# B&R Automation Studio project Lab2_Conveyor
Automation Studio 4.5.2.102; Conveyor station; technology packages: Acp10Arnc0 5.2.1, mapp 5.2.1

## Configuration Distributor

CPU 5PP5CP.US15-02, AutomationRuntime D4.52, Build 4.1.2, Vc V4.52.0

### Task classes (Cpu.sw)
```
Cyclic#1 (cycle 2000 us, tolerance 0 us):
  ncsdcctrl <- ncsdcctrl.prg
  IOCtrl1 <- (binary)
  IOCtrl <- (binary)
Cyclic#4:
  Ejector <- Distributing.Machine.Ejector.prg
  SwivelDriv <- Distributing.Machine.SwivelDrive.prg
  AlarmCtrl <- Distributing.AlarmCtrl.prg
  MainCtrl <- Distributing.Machine.MainCtrl.prg
  Conveyor <- Distributing.Machine.Conveyor.Conveyor.prg
  VisCtrl <- Distributing.Visualization.VisCtrl.prg [disabled]
DataObjects: Acp10sys
NcDataObjects: gAxisDista <- Distributing.Machine.Conveyor.gAxisDistobj.gAxisDista.dob, gAxisDisti <- Distributing.Machine.Conveyor.gAxisDistobj.gAxisDisti.dob, acp10etxen <- acp10etxen.dob
VcDataObjects: VisuDi <- Distributing.Visualization.VisuDist.dob
Binaries: udbdef, TCData, arsvcreg, vccdt, vccbmp, vcfile, arial, vcrt, vcbclass, vccbtn, vcmgr, vcgclass, vcdsint, vcnet, vcptelo, vccline, vcpdihd, vcpfpp50, vcshared, vcclbox, vccscale, arialbd, vccnum, vcpdvnc, vcpdi855, vcpdsw, VisuDi01, vccshape, VisuDi02, vcctext, vcfntttf, vccovl, vcalarm, vcpdi815, VisuDi03, vcdsloc, vcpfmtcx, vctcal, arconfig, User, Config, ashwd, sysconf, ashwac, Role, asfw, iomap, OpcUaMap, Acp10map, acp10cfg
Libraries: AsOpcUac, runtime, AsOpcUas, asstring, brsystem, MpBase, MpCom, standard, sys_lib, Acp10par, NcGlobal, Acp10man, Acp10sdc, Acp10_MC, AsBrStr, MpAxis, asieccon, fileio, astime, dataobj, powerlnk, vcresman
```

### Hardware
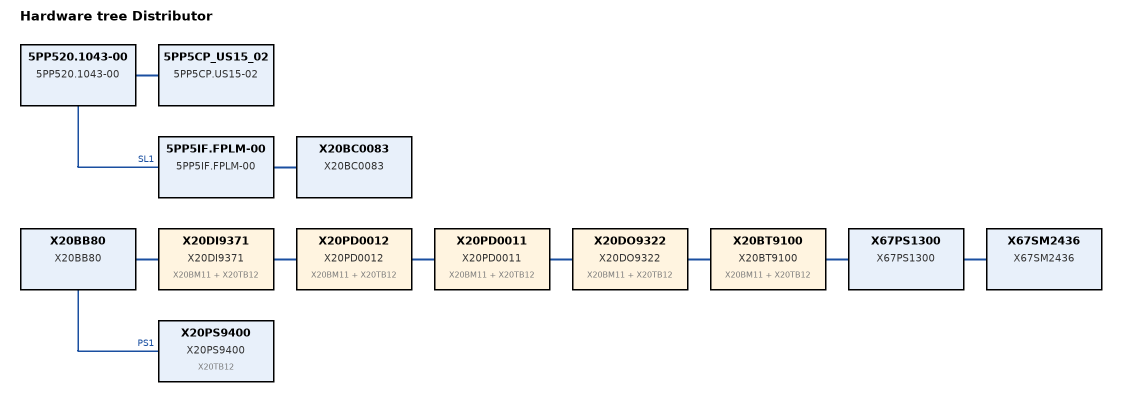
```
5PP520.1043-00 : 5PP520.1043-00 v2.0.3.1
  Connector IF3:
    ActivateDevice = 1
    Mode = Manual
    InternetAddress = 10.10.10.99
    SubnetMask = 255.255.255.0
    Vnc1
    VncVcObjectName1 = VisuDi
    VncKeyMappingFile1 = 
    VncRefreshRate1 = 250
  VcObjectName = VisuDi
5PP5CP_US15_02 : 5PP5CP.US15-02 v2.0.6.0  [SY -> 5PP520.1043-00.SY1]
  ConfigurationID = Lab2_Conveyor_Distributor
  TimerDeviceType = EPLX2X
  TimerDevice = 5PP5IF.FPLM-00.IF1
  TaskClassIdleTime = 2000
  Cyclic1Duration = 2000
  Cyclic1Tolerance = 0
  Cyclic1Output = 1
  ActivateOpcUa = 1
  OpcUaInformationModels_PV_Version = 1
5PP5IF.FPLM-00 : 5PP5IF.FPLM-00 v2.4.0.0  [SL -> 5PP520.1043-00.SL1]
X20BB80 : X20BB80 v1.0.2.0
X20BC0083 : X20BC0083 v2.7.0.0  [PLK1 -> 5PP5IF.FPLM-00.IF1 (NodeNumber=2) [Cable Type=PowerlinkCable, Length=10, Version=1.0.0.2]; SL -> X20BB80.SL1]
  Supervision = off
X20BM11 : X20BM11 v1.0.0.1  [X2X1 -> X20BB80.IF1]
X20BM11a : X20BM11 v1.0.0.1  [X2X1 -> X20BM11.X2X2]
X20BM11b : X20BM11 v1.0.0.1  [X2X1 -> X20BM11a.X2X2]
X20BM11c : X20BM11 v1.0.0.1  [X2X1 -> X20BM11b.X2X2]
X20BM11d : X20BM11 v1.0.0.1  [X2X1 -> X20BM11c.X2X2]
X20BT9100 : X20BT9100 v1.0.3.0  [SS1 -> X20TB12e.SS; SL -> X20BM11d.SL1]
  Supervision = off
X20DI9371 : X20DI9371 v1.0.2.0  [SS1 -> X20TB12a.SS; SL -> X20BM11.SL1]
  Supervision = off
X20DO9322 : X20DO9322 v1.0.3.0  [SS1 -> X20TB12d.SS; SL -> X20BM11c.SL1]
  Supervision = off
X20PD0011 : X20PD0011 v1.0.2.0  [SS1 -> X20TB12c.SS; SL -> X20BM11b.SL1]
  Supervision = off
X20PD0012 : X20PD0012 v1.0.2.0  [SS1 -> X20TB12b.SS; SL -> X20BM11a.SL1]
  Supervision = off
X20PS9400 : X20PS9400 v1.0.2.4  [SS1 -> X20TB12.SS; PS -> X20BB80.PS1]
  Supervision = off
X20TB12 : X20TB12 v1.0.0.0
X20TB12a : X20TB12 v1.0.0.0
X20TB12b : X20TB12 v1.0.0.0
X20TB12c : X20TB12 v1.0.0.0
X20TB12d : X20TB12 v1.0.0.0
X20TB12e : X20TB12 v1.0.0.0
X67PS1300 : X67PS1300 v1.0.0.0  [X2X1 -> X20BT9100.X2X1 [Cable Type=X2XCable, Length=10, Version=1.0.0.2]]
X67SM2436 : X67SM2436 v1.5.0.1  [X2X1 -> X67PS1300.X2X2 [Cable Type=X2XCable, Length=10, Version=1.0.0.2]]
  Supervision = off
  HoldingCurrent01 = 0
  RatedCurrent01 = 100
  MaximumCurrent01 = 160
  LatchSync01 = Stepper 1 latch value synchron (AB/R_1 latch value asynchron)
  LatchSync02 = Stepper 2 latch value synchron (AB/R_2 latch value asynchron)
  SCALE_ENCOD_INCR_r1 = 51200
  BothEndSwitchesAreNormallyOpen_r1 = on
```

### IoMap.iom - 5PP5CP_US15_02/IoMap.iom
```iecst
VAR_CONFIG
	Cyclic#1.gAxisDist_DrvIf.iLifeCnt AT %IB."X67SM2436".LifeCnt;
	Cyclic#1.gAxisDist_DrvIf.iDrvOK AT %IX."X67SM2436".DrvOk01;
	Cyclic#1.gAxisDist_DrvIf.oBoostCurrent AT %QX."X67SM2436".BoostCurrent01;
	Cyclic#1.gAxisDist_DrvIf.oStandStillCurrent AT %QX."X67SM2436".StandstillCurrent01;
	Cyclic#1.gAxisDist_DrvIf.oSetTime AT %QW."X67SM2436".SetTime01;
	Cyclic#1.gAxisDist_MotorStep0 AT %QW."X67SM2436".Motor1Step0;
	Cyclic#1.gAxisDist_DiDoIf.iLifeCntDriveEnable AT %IB."X67SM2436".LifeCnt;
	Cyclic#1.gAxisDist_DiDoIf.iLifeCntDriveReady AT %IB."X67SM2436".LifeCnt;
	Cyclic#1.gAxisDist_DiDoIf.iDriveReady AT %IX."X67SM2436".DrvOk01;
	Cyclic#1.gAxisDist_DiDoIf.oDriveEnable AT %QX."X67SM2436".DriveEnable01;
	Cyclic#1.gAxisDist_EncIf1.iLifeCnt AT %IB."X67SM2436".LifeCnt;
	Cyclic#1.gAxisDist_EncIf1.iEncOK AT %IX."X67SM2436".EncOk01;
	Cyclic#1.gAxisDist_EncIf1.iActPos AT %IW."X67SM2436".ActPos01;
	Cyclic#1.gAxisDist_EncIf1.iRefPulsePos AT %IW."X67SM2436".RefPulsePos01;
	Cyclic#1.gAxisDist_EncIf1.iRefPulseCnt AT %IB."X67SM2436".RefPulseCnt01;
	Cyclic#1.gAxisDist_EncIf1.iActTime AT %IW."X67SM2436".ActTime01;
	::gDistModuleOK.Interface AT %IX."5PP5IF.FPLM-00".ModuleOk;
	::gDistModuleOK.BusController AT %IX."X20BC0083".ModuleOk;
	::gDistModuleOK.PowerSupply AT %IX."X20PS9400".ModuleOk;
	::gDistModuleOK.DigitalInput AT %IX."X20DI9371".ModuleOk;
	::gDistModuleOK.PotentialDist0012 AT %IX."X20PD0012".ModuleOk;
	::gDistModuleOK.PotentialDist0011 AT %IX."X20PD0011".ModuleOk;
	::gDistModuleOK.DigitalOutput AT %IX."X20DO9322".ModuleOk;
	::gDistModuleOK.BusTransmitter AT %IX."X20BT9100".ModuleOk;
	::gDistModuleOK.StepperMotor AT %IX."X67SM2436".ModuleOk;
	::gDistHW.di.ProductGripped AT %IX."X20DI9371".DigitalInput04; (* *) (*Product gripped with suction*)
	::gDistHW.di.SwDrMagPos AT %IX."X20DI9371".DigitalInput05; (* *) (*Swivel drive in magazine position*)
	::gDistHW.di.SwDrConvPos AT %IX."X20DI9371".DigitalInput06; (* *) (*Swivel drive in conveyor position*)
	::gDistHW.di.MagEmpty AT %IX."X20DI9371".DigitalInput07; (* *) (*Magazine empty*)
	::gDistHW.di.SortStationFree AT %IX."X20DI9371".DigitalInput08; (* *) (*Sorting station free*)
	::gDistHW.do.EjCylPushProduct AT %QX."X20DO9322".DigitalOutput01; (* *) (*Ejecting cylinder push out product*)
	::gDistHW.do.Vacuum AT %QX."X20DO9322".DigitalOutput02; (* *) (*Vacuum on swivel drive*)
	::gDistHW.do.EjImpulse AT %QX."X20DO9322".DigitalOutput03; (* *) (*Ejection impulse on swivel drive*)
	::gDistHW.do.SwDrToMag AT %QX."X20DO9322".DigitalOutput04; (* *) (*Swivel drive to magazine*)
	::gDistHW.do.SwDrToConv AT %QX."X20DO9322".DigitalOutput05; (* *) (*Swivel drive to conveyor*)
	::gDistHW.di.EjCylRetracted AT %IX."X20DI9371".DigitalInput02; (* *) (*Ejecting cylinder retracted*)
	::gDistHW.di.EjCylExtended AT %IX."X20DI9371".DigitalInput03; (* *) (*Ejecting cylinder extended*)
	::gDistHW.di.PuckAtConvEnd AT %IX."X67SM2436".StatusInput01; (*Logical condition digital input 2, ABR2-A*) (*Conveyor - product on unloading position*) (*Logical condition digital input 4, ABR2-A*)
	::gDistHW.di.ConvStartVacant AT %IX."X67SM2436".StatusInput02; (*Logical condition digital input 1, ABR1-A*) (*Conveyor - product on starting position*)
END_VAR
```

### Acp10cfg.ncc - 5PP5CP_US15_02/Motion/Acp10cfg.ncc
```
NcConfiguration (Version=5.02.1, NcSwId=Acp10)
  ACP10CF1_typ:
    cnt_nettrc_rec_drive = 65535
    bufsize_trace_upload = 1200
    tc_nc_man_task = Cyclic #1
    glob_pv_as_ncobject = Yes
    ncsys_dl_broadcast = Yes
    ncsys_dl_acp_reset = Yes
    safemc_log_err_to_ax = Yes
    network_init:
      ncsw_init_execute = Yes
      automatic_execute = No
      node_nr_warning = Yes
      net_err_before_ncact = Yes
    nettrc:
      enter_parsecrec = Yes
      enter_ncaction = Yes
      save_ring_startidx = No
    cam_prof_download:
      cam_dat_dl_parallel = No
      tc_cam_dl_parallel = Task class for NC Manager task
    sdc_if[0]:
      if_name = SDC_IF1
      mc_broadcast_size = 800
      mc_broadcast_extdat = No
```

### Acp10map.ncm - 5PP5CP_US15_02/Motion/Acp10map.ncm
```
NcMapping (NcSwId=Acp10)
  NcObject gAxisDist (ModuleId=X67SM2436, ModuleAddress=SDC_IF1.ST1, Type=ncAXIS, Channel=1, AcoposSimulation=Off, InitParameter=gAxisDisti, AcoposParameter=gAxisDista, Disabled=FALSE, ModuleDisabled=FALSE)
  NcObject X67SM2436_ncAXIS2 (ModuleId=X67SM2436, ModuleAddress=SDC_IF1.ST2, Type=ncAXIS, Channel=1, AcoposSimulation=Off, Disabled=TRUE, ModuleDisabled=FALSE)
```

### Config.mpaxisbasic - 5PP5CP_US15_02/Motion/Config.mpaxisbasic
```
Element gAxisBasic (Type=mpaxisbasic)
  AxisConfiguration = AxisWithConfiguration
    Axis:
      BaseType = 2
      MeasurementUnit = 1
      PeriodSettings:
        Period = 108.0
      MovementLimits:
        VelocityPositive = 5000.0
        VelocityNegative = 5000.0
        Acceleration = 10000.0
        Deceleration = 10000.0
    Drive:
      Transformation:
        ReferenceDistance = 108.0
      Controller:
        LoopFilters:
          [0]
          [1]
          [2]
```

### Config_1.mpalarmxcore - 5PP5CP_US15_02/mappServices/Config_1.mpalarmxcore
```
Element gAlarmXCore_Dist (Type=mpalarmxcore)
  mapp.AlarmX.Core:
    Mapping:
      [0]:
        Alarm = Ejector Station - Cylinder Blocked
        [0] = Reaction
          Name = ErrorReaction
      [1]:
        Alarm = Swivel Arm - Motion Blocked
        [0] = Reaction
          Name = ErrorReaction
      [2]:
        Alarm = Conveyor - Puck Lost
        [0] = Reaction
          Name = ErrorReaction
      [3]:
        Alarm = Conveyor - Product Backlog
        [0] = Reaction
          Name = ErrorReaction
  mapp.AlarmX.Core.Configuration:
    [0]:
      Name = Ejector Station - Cylinder Blocked
      Message = Check for a backup in the ejector tray or a puck jammed in the magazine.
    [1]:
      Name = Swivel Arm - Motion Blocked
      Message = The Swivel Arm could not reach the requested position. Check for blockages.
    [2]:
      Name = Conveyor - Puck Lost
      Message = A puck is taking too long to reach the conveyor's end. Check for a lost puck or a sideways puck on the conveyor.
    [3]:
      Name = Conveyor - Product Backlog
      Message = There are too many unsorted pucks on the conveyor. Please remove excess pucks.
```

### Config_2.mpalarmxhistory - 5PP5CP_US15_02/mappServices/Config_2.mpalarmxhistory
```
Element gAlarmXHistory_Dist (Type=mpalarmxhistory)
```

## Configuration Sorter

CPU 5PP5CP.US15-02, AutomationRuntime D4.52, Build 4.1.2, Vc V4.52.0

### Task classes (Cpu.sw)
```
Cyclic#1 (cycle 2000 us, tolerance 0 us):
  ncsdcctrl <- ncsdcctrl.prg
Cyclic#4:
  MainCtrl <- Sorting.Machine.MainCtrl.prg
  OPCUAClien <- Sorting.OPCUA.OPCUAClient.prg [disabled]
  OPCUAConne <- Sorting.OPCUA.OPCUAConnect.prg [disabled]
  IOCtrl <- Sorting.Machine.IOCtrl.prg
  SortingSta <- Sorting.Machine.SortingStation.prg
  AlarmCtrl <- Sorting.AlarmCtrl.prg
  VisCtrl <- Sorting.Visualization.VisCtrl.prg
DataObjects: Acp10sys
NcDataObjects: gAxisSorta <- Sorting.gAxisSortobj.gAxisSorta.dob, gAxisSorti <- Sorting.gAxisSortobj.gAxisSorti.dob, acp10etxen <- acp10etxen.dob
VcDataObjects: VisuSo <- Sorting.Visualization.VisuSort.dob
Binaries: TCData, udbdef, vccdt, VisuSo02, vccbmp, vcfile, arial, vcrt, vcbclass, vccbtn, vcmgr, vcgclass, vcdsint, vcnet, vcptelo, vccline, vcpdihd, vcpfpp50, vcshared, vcclbox, vccscale, arialbd, vccnum, vcpdvnc, vcpdi855, vcpdsw, vccshape, vcctext, vcfntttf, vccovl, vcalarm, vcpdi815, arsvcreg, vcdsloc, vcpfmtcx, vctcal, VisuSo01, VisuSo03, vcchspot, Config_2, Config_1, OpcUaMap, ashwd, Role, User, sysconf, ashwac, asfw, arconfig, Config, iomap, Acp10map, acp10cfg, vcpkat, vcpfar00
Libraries: Acp10sdc, Acp10man, Acp10_MC, sys_lib, brsystem, AsBrStr, operator, runtime, astime, AsIecCon, AsOpcUac, AsOpcUas, asstring, MpCom, MpBase, standard, Acp10par, NcGlobal, MpAxis, MpAlarmX, fileio, powerlnk, vcresman, dataobj, areventlog
```

### Hardware
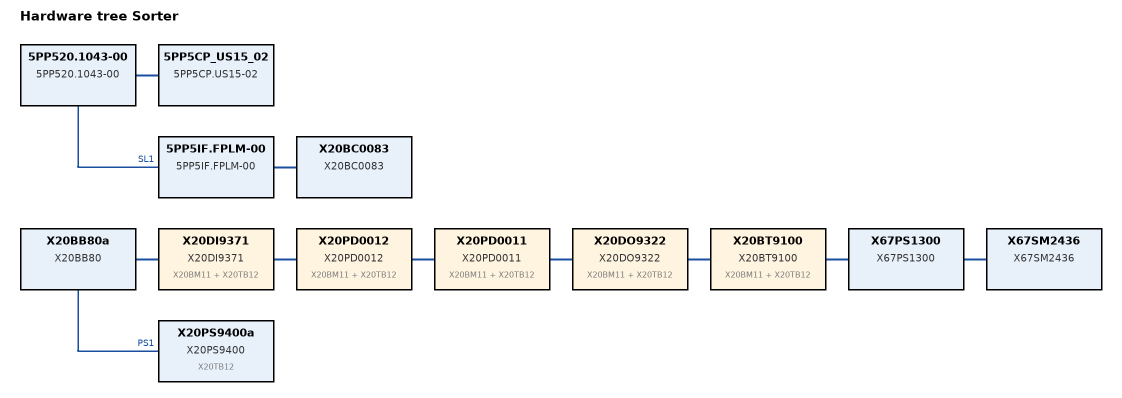
```
5PP520.1043-00 : 5PP520.1043-00 v2.0.3.1
  Connector IF3:
    ActivateDevice = 1
    Mode = Manual
    InternetAddress = 10.10.10.100
    SubnetMask = 255.255.255.0
    Vnc1
    VncVcObjectName1 = VisuSo
    VncKeyMappingFile1 = 
    VncRefreshRate1 = 250
  VcObjectName = VisuSo
5PP5CP_US15_02 : 5PP5CP.US15-02 v2.0.6.0  [SY -> 5PP520.1043-00.SY1]
  ConfigurationID = Lab2_Conveyor_Sorter
  TimerDeviceType = EPLX2X
  TimerDevice = 5PP5IF.FPLM-00.IF1
  TaskClassIdleTime = 2000
  Cyclic1Duration = 2000
  Cyclic1Tolerance = 0
  Cyclic1Output = 1
  ActivateOpcUa = 1
  OpcUaInformationModels_PV_Version = 1
5PP5IF.FPLM-00 : 5PP5IF.FPLM-00 v2.4.0.0  [SL -> 5PP520.1043-00.SL1]
X20BB80a : X20BB80 v1.0.2.0
X20BC0083 : X20BC0083 v2.7.0.0  [PLK1 -> 5PP5IF.FPLM-00.IF1 [Cable Type=PowerlinkCable, Length=10, Version=1.0.0.2]; SL -> X20BB80a.SL1]
X20BM11 : X20BM11 v1.0.0.1  [X2X1 -> X20BB80a.IF1]
X20BM11a : X20BM11 v1.0.0.1  [X2X1 -> X20BM11.X2X2]
X20BM11b : X20BM11 v1.0.0.1  [X2X1 -> X20BM11a.X2X2]
X20BM11c : X20BM11 v1.0.0.1  [X2X1 -> X20BM11b.X2X2]
X20BM11d : X20BM11 v1.0.0.1  [X2X1 -> X20BM11c.X2X2]
X20BT9100 : X20BT9100 v1.0.3.0  [SS1 -> X20TB12e.SS; SL -> X20BM11d.SL1]
X20DI9371 : X20DI9371 v1.0.2.0  [SS1 -> X20TB12b.SS; SL -> X20BM11.SL1]
X20DO9322 : X20DO9322 v1.0.3.0  [SS1 -> X20TB12d.SS; SL -> X20BM11c.SL1]
X20PD0011 : X20PD0011 v1.0.2.0  [SS1 -> X20TB12c.SS; SL -> X20BM11b.SL1]
X20PD0012 : X20PD0012 v1.0.2.0  [SS1 -> X20TB12.SS; SL -> X20BM11a.SL1]
X20PS9400a : X20PS9400 v1.0.2.4  [SS1 -> X20TB12a.SS; PS -> X20BB80a.PS1]
X20TB12 : X20TB12 v1.0.0.0
X20TB12a : X20TB12 v1.0.0.0
X20TB12b : X20TB12 v1.0.0.0
X20TB12c : X20TB12 v1.0.0.0
X20TB12d : X20TB12 v1.0.0.0
X20TB12e : X20TB12 v1.0.0.0
X67PS1300 : X67PS1300 v1.0.0.0  [X2X1 -> X20BT9100.X2X1 [Cable Type=X2XCable, Length=10, Version=1.0.0.2]]
X67SM2436 : X67SM2436 v1.5.0.1  [X2X1 -> X67PS1300.X2X2 [Cable Type=X2XCable, Length=10, Version=1.0.0.2]]
  Supervision = off
  HoldingCurrent01 = 0
  RatedCurrent01 = 80
  MaximumCurrent01 = 160
  LatchSync01 = Stepper 1 latch value synchron (AB/R_1 latch value asynchron)
  SCALE_ENCOD_INCR_r1 = 51200
```

### IoMap.iom - 5PP5CP_US15_02/IoMap.iom
```iecst
VAR_CONFIG
	Cyclic#1.gAxisSort_DrvIf.iLifeCnt AT %IB."X67SM2436".LifeCnt;
	Cyclic#1.gAxisSort_DrvIf.iDrvOK AT %IX."X67SM2436".DrvOk01;
	Cyclic#1.gAxisSort_DrvIf.oBoostCurrent AT %QX."X67SM2436".BoostCurrent01;
	Cyclic#1.gAxisSort_DrvIf.oStandStillCurrent AT %QX."X67SM2436".StandstillCurrent01;
	Cyclic#1.gAxisSort_DrvIf.oSetTime AT %QW."X67SM2436".SetTime01;
	Cyclic#1.gAxisSort_MotorStep0 AT %QW."X67SM2436".Motor1Step0;
	Cyclic#1.gAxisSort_DiDoIf.iLifeCntDriveEnable AT %IB."X67SM2436".LifeCnt;
	Cyclic#1.gAxisSort_DiDoIf.iLifeCntDriveReady AT %IB."X67SM2436".LifeCnt;
	Cyclic#1.gAxisSort_DiDoIf.iDriveReady AT %IX."X67SM2436".DrvOk01;
	Cyclic#1.gAxisSort_DiDoIf.oDriveEnable AT %QX."X67SM2436".DriveEnable01;
	Cyclic#1.gAxisSort_EncIf1.iLifeCnt AT %IB."X67SM2436".LifeCnt;
	Cyclic#1.gAxisSort_EncIf1.iEncOK AT %IX."X67SM2436".EncOk01;
	Cyclic#1.gAxisSort_EncIf1.iActPos AT %IW."X67SM2436".ActPos01;
	Cyclic#1.gAxisSort_EncIf1.iRefPulsePos AT %IW."X67SM2436".RefPulsePos01;
	Cyclic#1.gAxisSort_EncIf1.iRefPulseCnt AT %IB."X67SM2436".RefPulseCnt01;
	Cyclic#1.gAxisSort_EncIf1.iActTime AT %IW."X67SM2436".ActTime01;
	::gSortHW.do.ExtendSwitch1 AT %QX."X20DO9322".DigitalOutput02; (* *) (*Extend switch 1*)
	::gSortHW.do.ExtendSwitch2 AT %QX."X20DO9322".DigitalOutput03; (* *) (*Extend switch 2*)
	::gSortHW.do.RetractStopper AT %QX."X20DO9322".DigitalOutput04; (* *) (*Retract stopper*)
	::gSortHW.di.ProductAvailable AT %IX."X20DI9371".DigitalInput01; (* *) (*Product available*)
	::gSortHW.di.Metallic AT %IX."X20DI9371".DigitalInput02; (* *) (*Metallic product*)
	::gSortHW.di.NotBlack AT %IX."X20DI9371".DigitalInput03; (* *) (*Product is not black*)
	::gSortHW.di.LaneFull AT %IX."X20DI9371".DigitalInput04; (* *) (*Lane full*)
	::gSortHW.di.Switch1Retracted AT %IX."X20DI9371".DigitalInput05; (* *) (*Switch 1 retracted*)
	::gSortHW.di.Switch1Extended AT %IX."X20DI9371".DigitalInput06; (* *) (*Switch 1 extended*)
	::gSortHW.di.Switch2Retracted AT %IX."X20DI9371".DigitalInput07; (* *) (*Switch 2 retracted*)
	::gSortHW.di.Switch2Extended AT %IX."X20DI9371".DigitalInput08; (* *) (*Switch 2 extended*)
	::gSortModuleOK.Interface AT %IX."5PP5IF.FPLM-00".ModuleOk;
	::gSortModuleOK.BusController AT %IX."X20BC0083".ModuleOk;
	::gSortModuleOK.PowerSupply AT %IX."X20PS9400a".ModuleOk;
	::gSortModuleOK.DigitalInput AT %IX."X20DI9371".ModuleOk;
	::gSortModuleOK.PotentialDist0012 AT %IX."X20PD0012".ModuleOk;
	::gSortModuleOK.PotentialDist0011 AT %IX."X20PD0011".ModuleOk;
	::gSortModuleOK.DigitalOutput AT %IX."X20DO9322".ModuleOk;
	::gSortModuleOK.BusTransmitter AT %IX."X20BT9100".ModuleOk;
	::gSortModuleOK.StepperMotor AT %IX."X67SM2436".ModuleOk;
END_VAR
```

### Acp10cfg.ncc - 5PP5CP_US15_02/Motion/Acp10cfg.ncc
```
NcConfiguration (Version=5.02.1, NcSwId=Acp10)
  ACP10CF1_typ:
    cnt_nettrc_rec_drive = 65535
    bufsize_trace_upload = 1200
    tc_nc_man_task = Cyclic #1
    glob_pv_as_ncobject = Yes
    ncsys_dl_broadcast = Yes
    ncsys_dl_acp_reset = Yes
    safemc_log_err_to_ax = Yes
    network_init:
      ncsw_init_execute = Yes
      automatic_execute = No
      node_nr_warning = Yes
      net_err_before_ncact = Yes
    nettrc:
      enter_parsecrec = Yes
      enter_ncaction = Yes
      save_ring_startidx = Yes
    cam_prof_download:
      cam_dat_dl_parallel = No
      tc_cam_dl_parallel = Task class for NC Manager task
    sdc_if[0]:
      if_name = SDC_IF1
      mc_broadcast_size = 800
      mc_broadcast_extdat = No
```

### Acp10map.ncm - 5PP5CP_US15_02/Motion/Acp10map.ncm
```
NcMapping (NcSwId=Acp10, DisabledNodesAreHidden=False)
  NcObject gAxisSort (ModuleId=X67SM2436, ModuleAddress=SDC_IF1.ST1, Type=ncAXIS, Channel=1, AcoposSimulation=Off, InitParameter=gAxisSorti, AcoposParameter=gAxisSorta, Disabled=FALSE, ModuleDisabled=FALSE)
  NcObject X67SM2436_ncAXIS2 (ModuleId=X67SM2436, ModuleAddress=SDC_IF1.ST2, Type=ncAXIS, Channel=1, AcoposSimulation=Off, Disabled=TRUE, ModuleDisabled=FALSE)
```

### Config.mpaxisbasic - 5PP5CP_US15_02/Motion/Config.mpaxisbasic
```
Element gAxisBasic (Type=mpaxisbasic)
  AxisConfiguration = AxisWithConfiguration
    Axis:
      BaseType = 2
      MeasurementUnit = 1
      MeasurementResolution = 1
      PeriodSettings:
        Period = 150
      MovementLimits:
        VelocityPositive = 10000
        VelocityNegative = 10000
        Acceleration = 50000
        Deceleration = 50000
    Drive:
      Transformation:
        ReferenceDistance = 150
      Controller:
        LoopFilters:
          [0]
          [1]
          [2]
```

### Config_1.mpalarmxcore - 5PP5CP_US15_02/mappServices/Config_1.mpalarmxcore
```
Element gAlarmXCore_Sort (Type=mpalarmxcore)
  mapp.AlarmX.Core.Configuration:
    [0]:
      Name = Lane1Full
      Message = Lane 1 is full.
      Code = 1
    [1]:
      Name = Lane2Full
      Message = Lane 2 is full.
      Code = 2
    [2]:
      Name = Lane3Full
      Message = Lane 3 is full.
      Code = 3
    [3]:
      Name = NoProductAvail
      Message = There is no product available.
      Code = 4
    [4]:
      Name = SwitchStuck
      Message = The switch is stuck.
      Code = 5
    [5]:
      Name = PuckMissing
      Message = No product detected.
      Code = 6
    [6]:
      Name = Axis
      Message = Axis error.
      Code = 7
    [7]:
      Name = CheckHW
      Message = Hardware module not OK.
      Code = 8
    [8]:
      Name = CheckMachine
      Message = Machine error.
      Code = 9
```

### Config_2.mpalarmxhistory - 5PP5CP_US15_02/mappServices/Config_2.mpalarmxhistory
```
Element gAlarmXHistory_Sort (Type=mpalarmxhistory)
```

## Logical view

Binary libraries used (declarations not repeated): operator, runtime, astime, AsIecCon, AsOpcUac, AsOpcUas, asstring, brsystem, MpCom 5.02.1, standard, sys_lib, AsBrStr, MpAxis 1.65.0, MpBase 5.02.0, NcGlobal, Acp10_MC, Acp10man, Acp10par, Acp10sdc, MpAlarmX 5.02.1

### Global.var - Global variables
```iecst
VAR
	gAxisDist : ACP10AXIS_typ; (*Axis variable distributor*)
	gAxisDist_HW : SdcHwCfg_typ := (0); (*Axis variable distributor*)
	gAxisDist_DrvIf : SdcDrvIf16_typ := (0); (*Axis variable distributor*)
	gAxisDist_EncIf1 : SdcEncIf16_typ := (0); (*Axis variable distributor*)
	gAxisDist_DiDoIf : SdcDiDoIf_typ := (0); (*Axis variable distributor*)
	gAxisDist_MotorStep0 : INT := 0; (*Axis variable distributor*)
	gAxisSort : ACP10AXIS_typ; (*Axis variable sorter*)
	gAxisSort_HW : SdcHwCfg_typ := (0); (*Axis variable sorter*)
	gAxisSort_DrvIf : SdcDrvIf16_typ := (0); (*Axis variable sorter*)
	gAxisSort_EncIf1 : SdcEncIf16_typ := (0); (*Axis variable sorter*)
	gAxisSort_DiDoIf : SdcDiDoIf_typ := (0); (*Axis variable sorter*)
	gAxisSort_MotorStep0 : INT := 0; (*Axis variable sorter*)
END_VAR
```

### Program Logical/ncsdcctrl (IEC) - ncsdcctrl

#### ncsdcctrl.var
```iecst
VAR
	gAxisDist_oSetPosOld : INT := 0;
	gAxisSort_oSetPosOld : INT := 0;
END_VAR
```

#### ncsdcctrlCyclic.st
```iecst
PROGRAM _CYCLIC

(* ### BEGIN gAxisDist ### *)

(* life counter emulation of digital inputs *)
       gAxisDist_DiDoIf.iLifeCntReference := gAxisDist_DiDoIf.iLifeCntReference + 1;
       gAxisDist_DiDoIf.iLifeCntNegHwEnd  := gAxisDist_DiDoIf.iLifeCntNegHwEnd  + 1;
       gAxisDist_DiDoIf.iLifeCntPosHwEnd  := gAxisDist_DiDoIf.iLifeCntPosHwEnd  + 1;

(* default function model of ACOPOSmicro: convert absolute steps to delta steps - overflow save delta calculation *)
       gAxisDist_MotorStep0 := gAxisDist_DrvIf.oSetPos - gAxisDist_oSetPosOld;
       gAxisDist_oSetPosOld := gAxisDist_DrvIf.oSetPos;

(* ### END gAxisDist ### *)

(* ### BEGIN gAxisSort ### *)

(* life counter emulation of digital inputs *)
       gAxisSort_DiDoIf.iLifeCntReference := gAxisSort_DiDoIf.iLifeCntReference + 1;
       gAxisSort_DiDoIf.iLifeCntNegHwEnd  := gAxisSort_DiDoIf.iLifeCntNegHwEnd  + 1;
       gAxisSort_DiDoIf.iLifeCntPosHwEnd  := gAxisSort_DiDoIf.iLifeCntPosHwEnd  + 1;

(* default function model of ACOPOSmicro: convert absolute steps to delta steps - overflow save delta calculation *)
       gAxisSort_MotorStep0 := gAxisSort_DrvIf.oSetPos - gAxisSort_oSetPosOld;
       gAxisSort_oSetPosOld := gAxisSort_DrvIf.oSetPos;

(* ### END gAxisSort ### *)

END_PROGRAM
```

#### ncsdcctrlInit.st
```iecst
PROGRAM _INIT

(* ### BEGIN gAxisDist ### *)

(* initialize general interfaces *)
       gAxisDist.size := gAxisDist.size;
       gAxisDist_HW.DrvIf_Typ := ncSDC_DRVSM16;
       brsstrcpy( ADR(gAxisDist_HW.DrvIf_Name[0]), ADR('gAxisDist_DrvIf') );
       gAxisDist_HW.DiDoIf_Typ := ncSDC_DIDO;
       brsstrcpy( ADR(gAxisDist_HW.DiDoIf_Name[0]), ADR('gAxisDist_DiDoIf') );
       gAxisDist_HW.EncIf1_Typ := ncSDC_ENC16;
       brsstrcpy( ADR(gAxisDist_HW.EncIf1_Name[0]), ADR('gAxisDist_EncIf1') );
       gAxisDist_EncIf1.iLifeCnt := gAxisDist_EncIf1.iLifeCnt;

(* initialize old-value for delta step calculation *)
       gAxisDist_oSetPosOld := gAxisDist_DrvIf.oSetPos;

(* ### END gAxisDist ### *)

(* ### BEGIN gAxisSort ### *)

(* initialize general interfaces *)
       gAxisSort.size := gAxisSort.size;
       gAxisSort_HW.DrvIf_Typ := ncSDC_DRVSM16;
       brsstrcpy( ADR(gAxisSort_HW.DrvIf_Name[0]), ADR('gAxisSort_DrvIf') );
       gAxisSort_HW.DiDoIf_Typ := ncSDC_DIDO;
       brsstrcpy( ADR(gAxisSort_HW.DiDoIf_Name[0]), ADR('gAxisSort_DiDoIf') );
       gAxisSort_HW.EncIf1_Typ := ncSDC_ENC16;
       brsstrcpy( ADR(gAxisSort_HW.EncIf1_Name[0]), ADR('gAxisSort_EncIf1') );
       gAxisSort_EncIf1.iLifeCnt := gAxisSort_EncIf1.iLifeCnt;

(* initialize old-value for delta step calculation *)
       gAxisSort_oSetPosOld := gAxisSort_DrvIf.oSetPos;

(* ### END gAxisSort ### *)

END_PROGRAM
```


### Package Logical/Distributing - Distributor configuration

### DistGlobal.typ - Package global types
```iecst
TYPE
	gDistHW_type : 	STRUCT  (*Hardware IO types for distributor*)
		di : diDist_type; (*Digital inputs for distributor*)
		do : doDist_type; (*Digital outputs for distributor*)
	END_STRUCT;
	diDist_type : 	STRUCT  (*Digital inputs for distributor*)
		EjCylExtended : BOOL; (*Ejecting cylinder extended*)
		EjCylRetracted : BOOL; (*Ejecting cylinder retracted*)
		ProductGripped : BOOL; (*Product gripped with suction*)
		SwDrMagPos : BOOL; (*Swivel drive in magazine position*)
		SwDrConvPos : BOOL; (*Swivel drive in conveyor position*)
		MagEmpty : BOOL; (*Magazine empty*)
		SortStationFree : BOOL; (*Sorting station free*)
		ConvStartVacant : BOOL; (*Conveyor - product on starting position*)
		PuckAtConvEnd : BOOL; (*Conveyor - product on unloading position*)
	END_STRUCT;
	doDist_type : 	STRUCT  (*Digital outputs for distributor*)
		EjCylPushProduct : BOOL; (*Ejecting cylinder push out product*)
		Vacuum : BOOL; (*Vacuum on swivel drive*)
		EjImpulse : BOOL; (*Ejection impulse on swivel drive*)
		SwDrToMag : BOOL; (*Swivel drive to magazine*)
		SwDrToConv : BOOL; (*Swivel drive to conveyor*)
	END_STRUCT;
	gDistModuleOK_type : 	STRUCT  (*Distributor module statuses*)
		Interface : BOOL; (*5PP5IF.FPLM-00 status*)
		BusController : BOOL; (*X20BC0083 status*)
		PowerSupply : BOOL; (*X20PS9400 status*)
		DigitalInput : BOOL; (*X20DI9371 status*)
		PotentialDist0012 : BOOL; (*X20PD0012 status*)
		PotentialDist0011 : BOOL; (*X20PD0011 status*)
		DigitalOutput : BOOL; (*X20DO9322 status*)
		BusTransmitter : BOOL; (*X20BT9100 status*)
		StepperMotor : BOOL; (*X67SM2436 status*)
	END_STRUCT;
END_TYPE
```

### DistGlobal.var - Package global variables
```iecst
VAR
	gDistHW : gDistHW_type; (*Control variable for hardware IO types for distributor*)
	gDistModuleOK : gDistModuleOK_type; (*Control variable for distributor module statuses*)
END_VAR
```

- Visualisation Logical/Distributing/Visualization (not shown)

### Package Logical/Distributing/Machine - Distributing machine functionality

### Package Logical/Distributing/Machine/Conveyor - Contains conveyor task and relevant motion items

### Package Logical/Distributing/Machine/Conveyor/gAxisDistobj - gAxisDistobj

### Data object Logical/Distributing/Machine/Conveyor/gAxisDistobj/gAxisDista (Apt)

#### gAxisDista.apt
```
AcoposParameterTable:
  Root Parameters:
    64232 = 51200 (Name=SM_SCALE_STEP)
    64233 = 1000 (Name=SM_SCALE_LOAD_UNITS)
    64234 = 1 (Name=SM_SCALE_LOAD_MOTREV)
    230 = PCTRL_S_SET (Name=PCTRL_S_ACT_PARID)  // CTRL Position controller: Actual encoder position parameter ID
```

### Data object Logical/Distributing/Machine/Conveyor/gAxisDistobj/gAxisDisti (Ax)

#### gAxisDisti.ax
```
InitParameter (Version=5.02.1, NcSwId=Acp10)
  ACP10AXIS_typ:
    dig_in:
      level:
        reference = ncACTIV_HI
        pos_hw_end = ncACTIV_HI
        neg_hw_end = ncACTIV_HI
        trigger1 = ncACTIV_HI
        trigger2 = ncACTIV_HI
    encoder_if:
      parameter:
        count_dir = ncSTANDARD
        scaling:
          load:
            units = 1000
            rev_motor = 1
    limit:
      parameter:
        v_pos = 3000.0
        v_neg = 3000.0
        a1_pos = 6000.0
        a2_pos = 6000.0
        a1_neg = 6000.0
        a2_neg = 6000.0
        t_jolt = 0
        t_in_pos = 0
        pos_sw_end = 2000000000
        neg_sw_end = -2000000000
        ds_warning = 500
        ds_stop = 1000
        a_stop = 1.0e30
        dv_stop = 0
        dv_stop_mode = ncOFF
    controller:
      mode = ncPOSITION
      position:
        kv = 50
        tn = 0
        t_predict = 0.01
        t_total = 0.01
        p_max = 1.0e30
        i_max = 0
      speed:
        kv = 2.0
        tn = 0
        t_filter = 0.0
        isq_filter1:
          type = ncOFF
          a0 = 0.0
          a1 = 0.0
          b0 = 0.0
          b1 = 0.0
          b2 = 0.0
          c0_par_id = 0
          c1_par_id = 0
        isq_filter2:
          type = ncOFF
          a0 = 0.0
          a1 = 0.0
          b0 = 0.0
          b1 = 0.0
          b2 = 0.0
          c0_par_id = 0
          c1_par_id = 0
        isq_filter3:
          type = ncOFF
          a0 = 0.0
          a1 = 0.0
          b0 = 0.0
          b1 = 0.0
          b2 = 0.0
          c0_par_id = 0
          c1_par_id = 0
      uf:
        type = ncLINEAR + ncCORRECTION
        auto_config = ncMOTOR_PAR
        u0 = 0
        un = 0
        fn = 50.0
        k_f_slip = 0
      ff:
        torque_load = 0.0
        torque_pos = 0.0
        torque_neg = 0.0
        kv_torque = 0.0
        inertia = 0.0
        t_filter_a = 0.0
    move:
      stop:
        parameter[0]:
          decel_ramp = ncA_LIMIT
          controller = ncON
        parameter[1]:
          decel_ramp = ncA_LIMIT
          controller = ncON
        parameter[2]:
          decel_ramp = ncA_LIMIT
          controller = ncON
        parameter[3]:
          decel_ramp = ncA_LIMIT
          controller = ncON
        quickstop:
          decel_ramp = ncA_LIMIT
          t_jolt = 0
        drive_error:
          decel_ramp = ncA_LIMIT
      homing:
        parameter:
          s = 0
          v_switch = 5000
          v_trigger = 500
          a = 50000
          mode = ncDIRECT
          edge_sw = ncPOSITIVE
          start_dir = ncPOSITIVE
          trigg_dir = ncPOSITIVE
          ref_pulse = ncOFF
          fix_dir = ncOFF
          tr_s_block = 0
          torque_lim = 0
          ds_block = 0
          ds_stop = 0
      basis:
        parameter:
          v_pos = 5000
          v_neg = 5000
          a1_pos = 50000
          a2_pos = 50000
          a1_neg = 50000
          a2_neg = 50000
    message:
      text:
        parameter:
          format = ncBREAK
          columns = 80
          data_modul = acp10etxen
```

### Program Logical/Distributing/Machine/Conveyor/Conveyor (IEC)

#### Cyclic.ld - Cyclic code
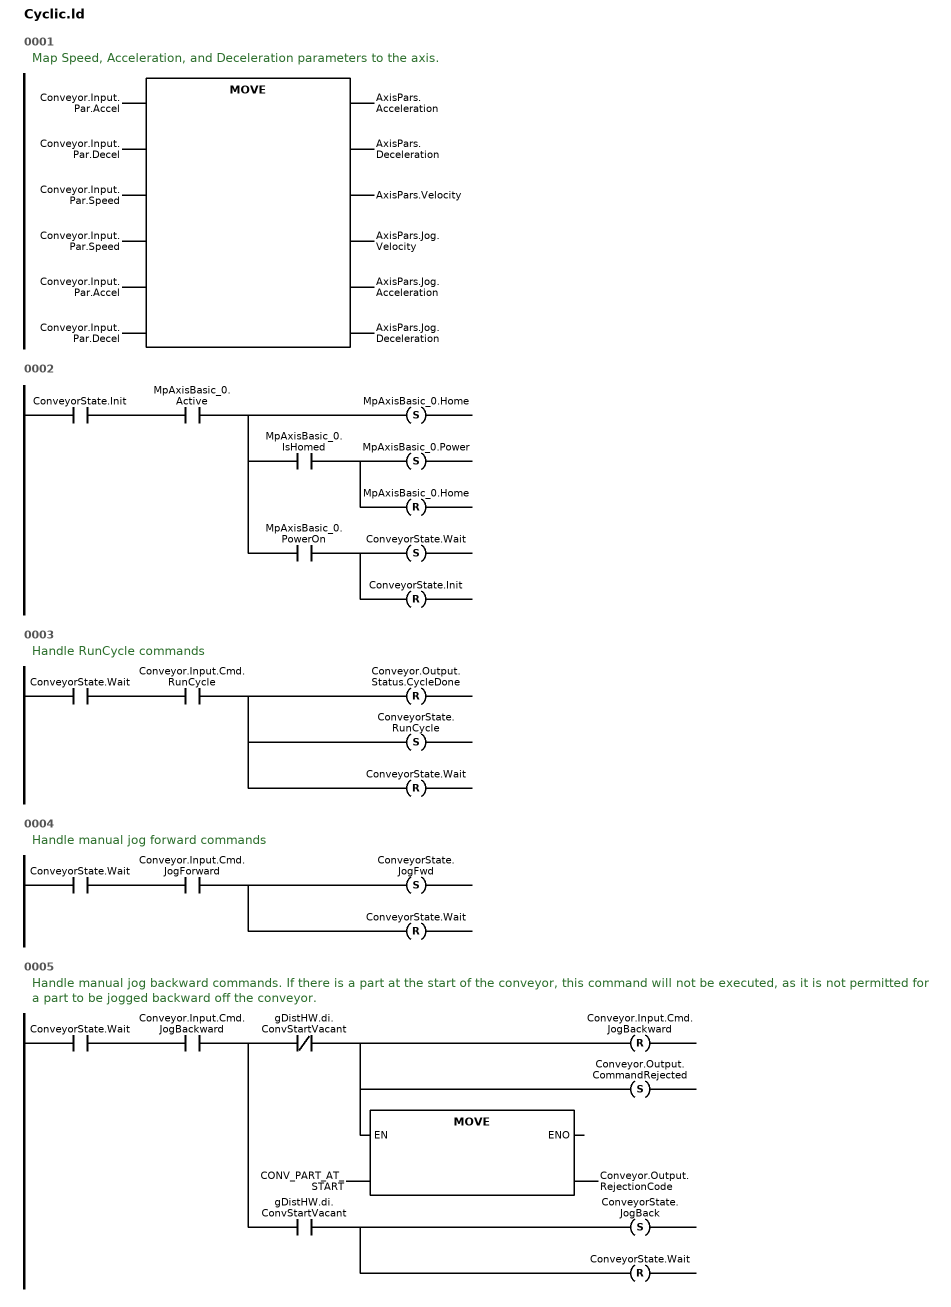
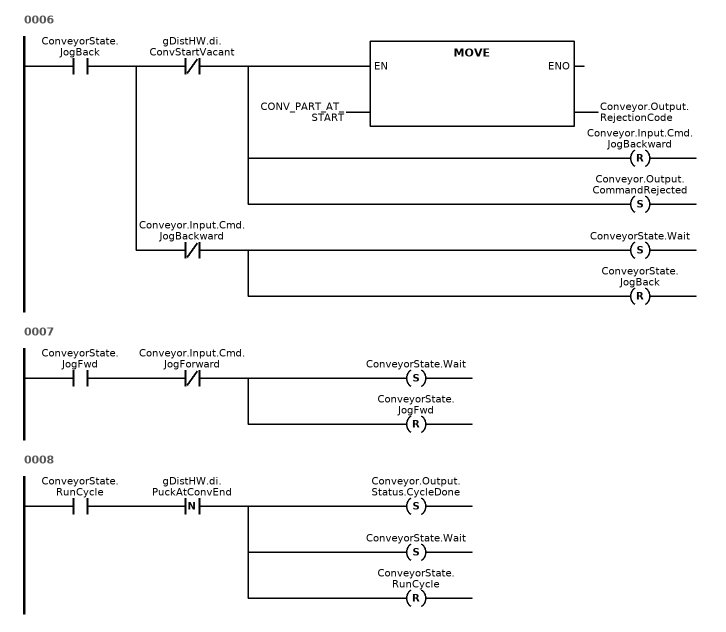
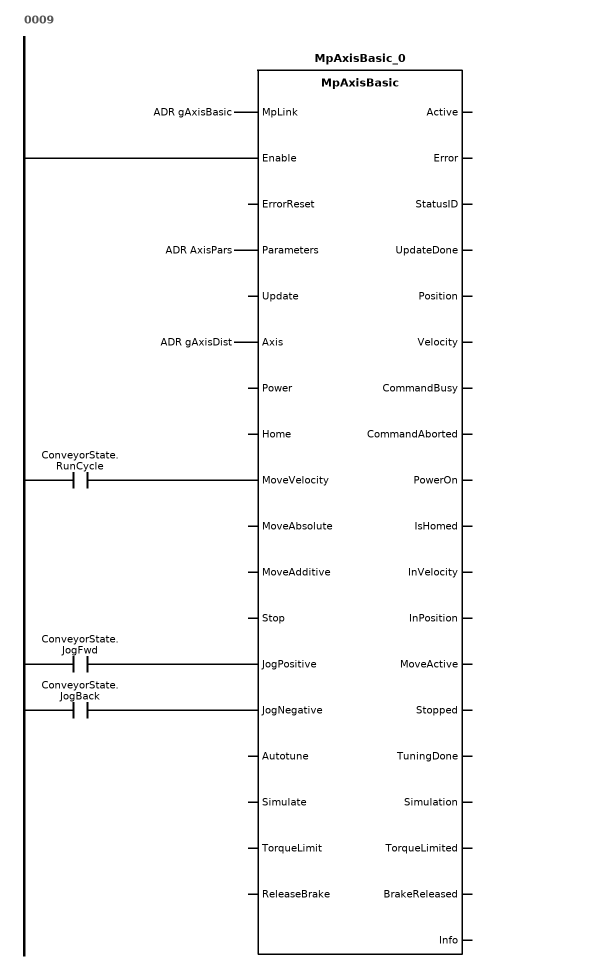
Ladder, written as Structured Text:
```iecst
(*********************************************************************************
 * Copyright:
 * Author:
 * Created:   	March 8, 2019/12:39 PM
 * Description:
 *********************************************************************************)
PROGRAM _CYCLIC
VAR
    _p1 : BOOL;
    _p2 : BOOL;
    _p3 : BOOL;
    _p4 : BOOL;
    _p5 : BOOL;
    _p6 : BOOL;
    _p7 : BOOL;
    _p8 : BOOL;
    _e9 : F_TRIG;
    _p10 : BOOL;
END_VAR
(* Network 1: Map Speed, Acceleration, and Deceleration parameters to the axis. *)
AxisPars.Acceleration := Conveyor.Input.Par.Accel;
AxisPars.Deceleration := Conveyor.Input.Par.Decel;
AxisPars.Velocity := Conveyor.Input.Par.Speed;
AxisPars.Jog.Velocity := Conveyor.Input.Par.Speed;
AxisPars.Jog.Acceleration := Conveyor.Input.Par.Accel;
AxisPars.Jog.Deceleration := Conveyor.Input.Par.Decel;

(* Network 2 *)
_p1 := ConveyorState.Init AND MpAxisBasic_0.Active;
IF ConveyorState.Init AND MpAxisBasic_0.Active THEN MpAxisBasic_0.Home := TRUE; END_IF;
_p2 := _p1 AND MpAxisBasic_0.IsHomed;
IF _p1 AND MpAxisBasic_0.IsHomed THEN MpAxisBasic_0.Power := TRUE; END_IF;
IF _p2 THEN MpAxisBasic_0.Home := FALSE; END_IF;
IF _p1 AND MpAxisBasic_0.PowerOn THEN
    ConveyorState.Wait := TRUE;
    ConveyorState.Init := FALSE;
END_IF;

(* Network 3: Handle RunCycle commands *)
_p3 := ConveyorState.Wait AND Conveyor.Input.Cmd.RunCycle;
IF _p3 THEN
    Conveyor.Output.Status.CycleDone := FALSE;
    ConveyorState.RunCycle := TRUE;
    ConveyorState.Wait := FALSE;
END_IF;

(* Network 4: Handle manual jog forward commands *)
_p4 := ConveyorState.Wait AND Conveyor.Input.Cmd.JogForward;
IF _p4 THEN
    ConveyorState.JogFwd := TRUE;
    ConveyorState.Wait := FALSE;
END_IF;

(* Network 5: Handle manual jog backward commands. If there is a part at the start of the conveyor, this command will not be executed, as it is not permitted for a part to be jogged backward off the conveyor. *)
_p5 := ConveyorState.Wait AND Conveyor.Input.Cmd.JogBackward;
IF _p5 AND NOT gDistHW.di.ConvStartVacant THEN
    Conveyor.Input.Cmd.JogBackward := FALSE;
    Conveyor.Output.CommandRejected := TRUE;
    Conveyor.Output.RejectionCode := CONV_PART_AT_START;
END_IF;
IF _p5 AND gDistHW.di.ConvStartVacant THEN
    ConveyorState.JogBack := TRUE;
    ConveyorState.Wait := FALSE;
END_IF;

(* Network 6 *)
_p6 := ConveyorState.JogBack AND NOT gDistHW.di.ConvStartVacant;
IF _p6 THEN
    Conveyor.Output.RejectionCode := CONV_PART_AT_START;
    Conveyor.Input.Cmd.JogBackward := FALSE;
    Conveyor.Output.CommandRejected := TRUE;
END_IF;
_p7 := ConveyorState.JogBack AND NOT Conveyor.Input.Cmd.JogBackward;
IF _p7 THEN
    ConveyorState.Wait := TRUE;
    ConveyorState.JogBack := FALSE;
END_IF;

(* Network 7 *)
_p8 := ConveyorState.JogFwd AND NOT Conveyor.Input.Cmd.JogForward;
IF _p8 THEN
    ConveyorState.Wait := TRUE;
    ConveyorState.JogFwd := FALSE;
END_IF;

(* Network 8 *)
_e9(CLK := gDistHW.di.PuckAtConvEnd);
IF ConveyorState.RunCycle AND _e9.Q THEN Conveyor.Output.Status.CycleDone := TRUE; END_IF;
_p10 := ConveyorState.RunCycle AND _e9.Q;
IF ConveyorState.RunCycle AND _e9.Q THEN ConveyorState.Wait := TRUE; END_IF;
IF _p10 THEN ConveyorState.RunCycle := FALSE; END_IF;

(* Network 9 *)
MpAxisBasic_0(MpLink := ADR(gAxisBasic), Enable := TRUE, Parameters := ADR(AxisPars), Axis := ADR(gAxisDist), MoveVelocity := ConveyorState.RunCycle, JogPositive := ConveyorState.JogFwd, JogNegative := ConveyorState.JogBack);
END_PROGRAM
```

#### Types.typ - Local data types
```iecst
TYPE
	ConveyorState_typ : 	STRUCT
		Init : BOOL := TRUE;
		Wait : BOOL := FALSE;
		RunCycle : BOOL := FALSE;
		JogFwd : BOOL := FALSE;
		JogBack : BOOL := FALSE;
		Error : BOOL := FALSE;
	END_STRUCT;
END_TYPE
```

#### Variables.var - Local variables
```iecst
VAR
	MpAxisBasic_0 : MpAxisBasic; (*Function block for MpAxisBasic*)
	ConveyorState : ConveyorState_typ;
	AxisPars : MpAxisBasicParType;
END_VAR
```

### Program Logical/Distributing/Machine/Conveyor/ncsdcctrl

#### ncsdcctrl.var
```iecst
VAR
	gAxisDist_oSetPosOld : INT := 0;
END_VAR
```

#### ncsdcctrlCyclic.st
```iecst
PROGRAM _CYCLIC

(* ### BEGIN gAxisDist ### *)

(* life counter emulation of digital inputs *)
       gAxisDist_DiDoIf.iLifeCntReference := gAxisDist_DiDoIf.iLifeCntReference + 1;
       gAxisDist_DiDoIf.iLifeCntNegHwEnd  := gAxisDist_DiDoIf.iLifeCntNegHwEnd  + 1;
       gAxisDist_DiDoIf.iLifeCntPosHwEnd  := gAxisDist_DiDoIf.iLifeCntPosHwEnd  + 1;

(* default function model of ACOPOSmicro: convert absolute steps to delta steps - overflow save delta calculation *)
       gAxisDist_MotorStep0 := gAxisDist_DrvIf.oSetPos - gAxisDist_oSetPosOld;
       gAxisDist_oSetPosOld := gAxisDist_DrvIf.oSetPos;

(* ### END gAxisDist ### *)

END_PROGRAM
```

#### ncsdcctrlInit.st
```iecst
PROGRAM _INIT

(* ### BEGIN gAxisDist ### *)

(* initialize general interfaces *)
       gAxisDist.size := gAxisDist.size;
       gAxisDist_HW.DrvIf_Typ := ncSDC_DRVSM16;
       brsstrcpy( ADR(gAxisDist_HW.DrvIf_Name[0]), ADR('gAxisDist_DrvIf') );
       gAxisDist_HW.DiDoIf_Typ := ncSDC_DIDO;
       brsstrcpy( ADR(gAxisDist_HW.DiDoIf_Name[0]), ADR('gAxisDist_DiDoIf') );
       gAxisDist_HW.EncIf1_Typ := ncSDC_ENC16;
       brsstrcpy( ADR(gAxisDist_HW.EncIf1_Name[0]), ADR('gAxisDist_EncIf1') );
       gAxisDist_EncIf1.iLifeCnt := gAxisDist_EncIf1.iLifeCnt;

(* initialize old-value for delta step calculation *)
       gAxisDist_oSetPosOld := gAxisDist_DrvIf.oSetPos;

(* ### END gAxisDist ### *)

END_PROGRAM
```

### Program Logical/Distributing/Machine/MainCtrl1 (IEC) - Distributing main control

#### Cyclic.ld - Cyclic code
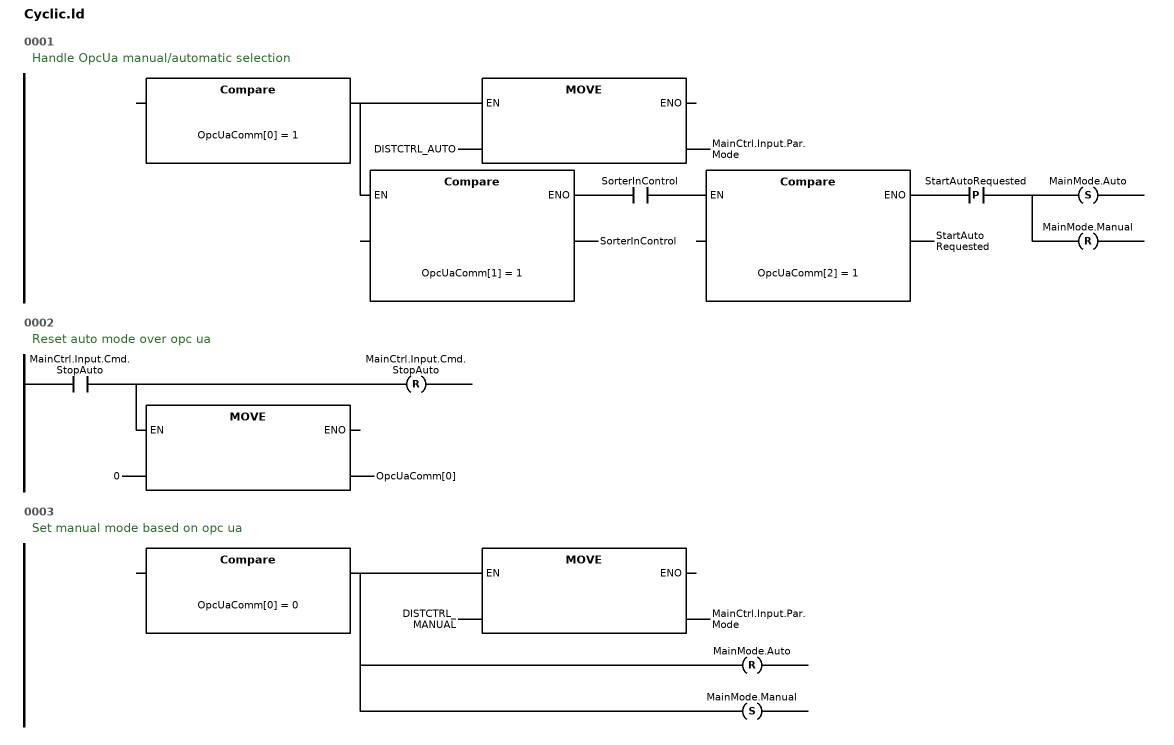
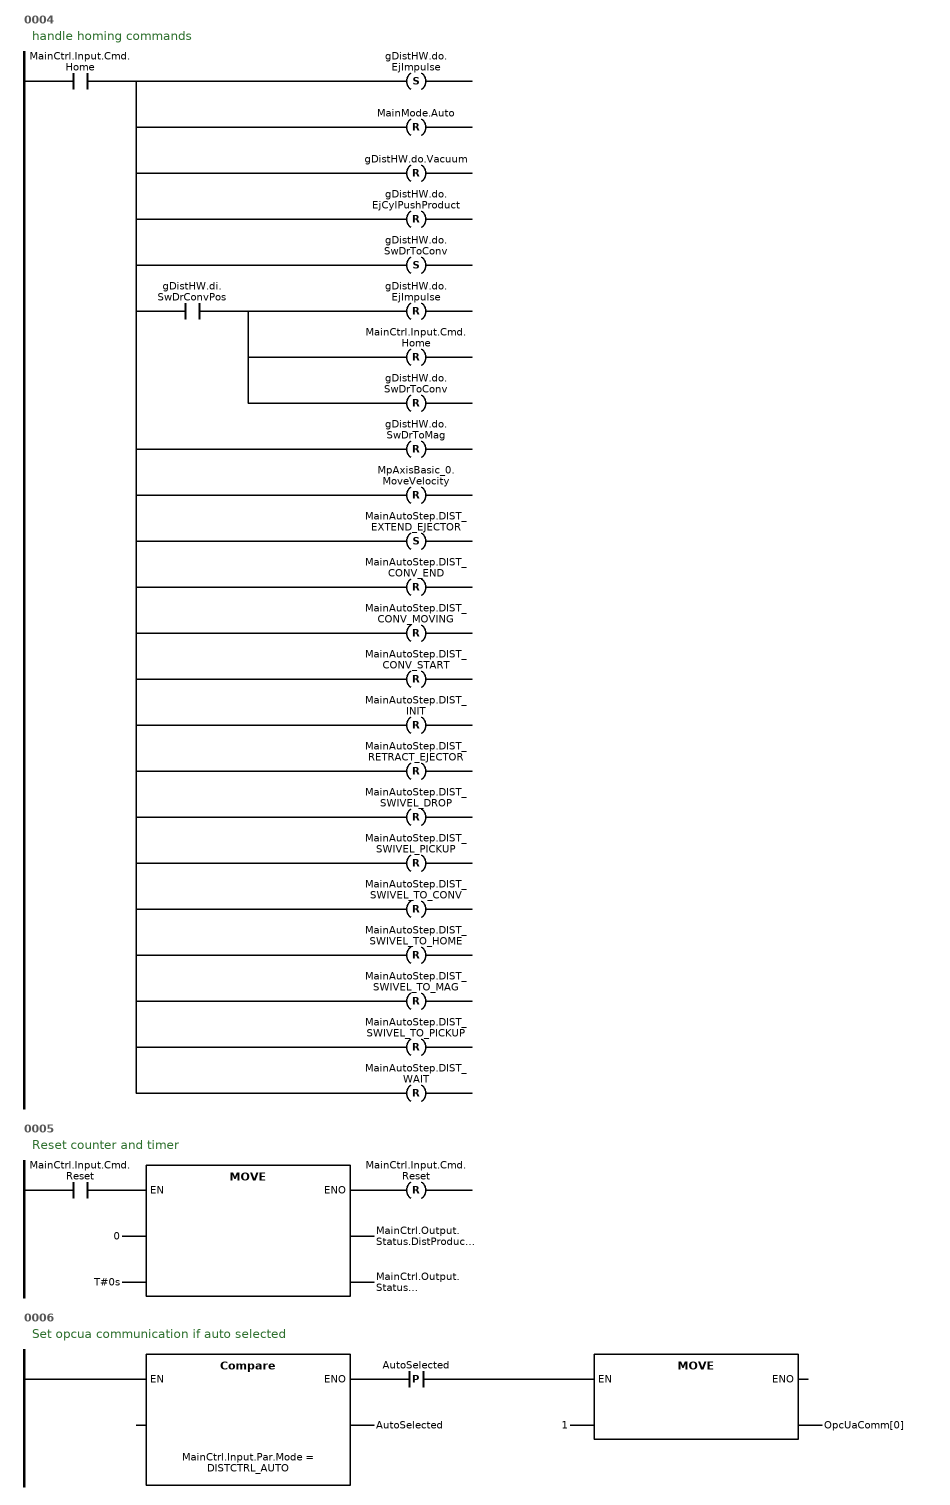
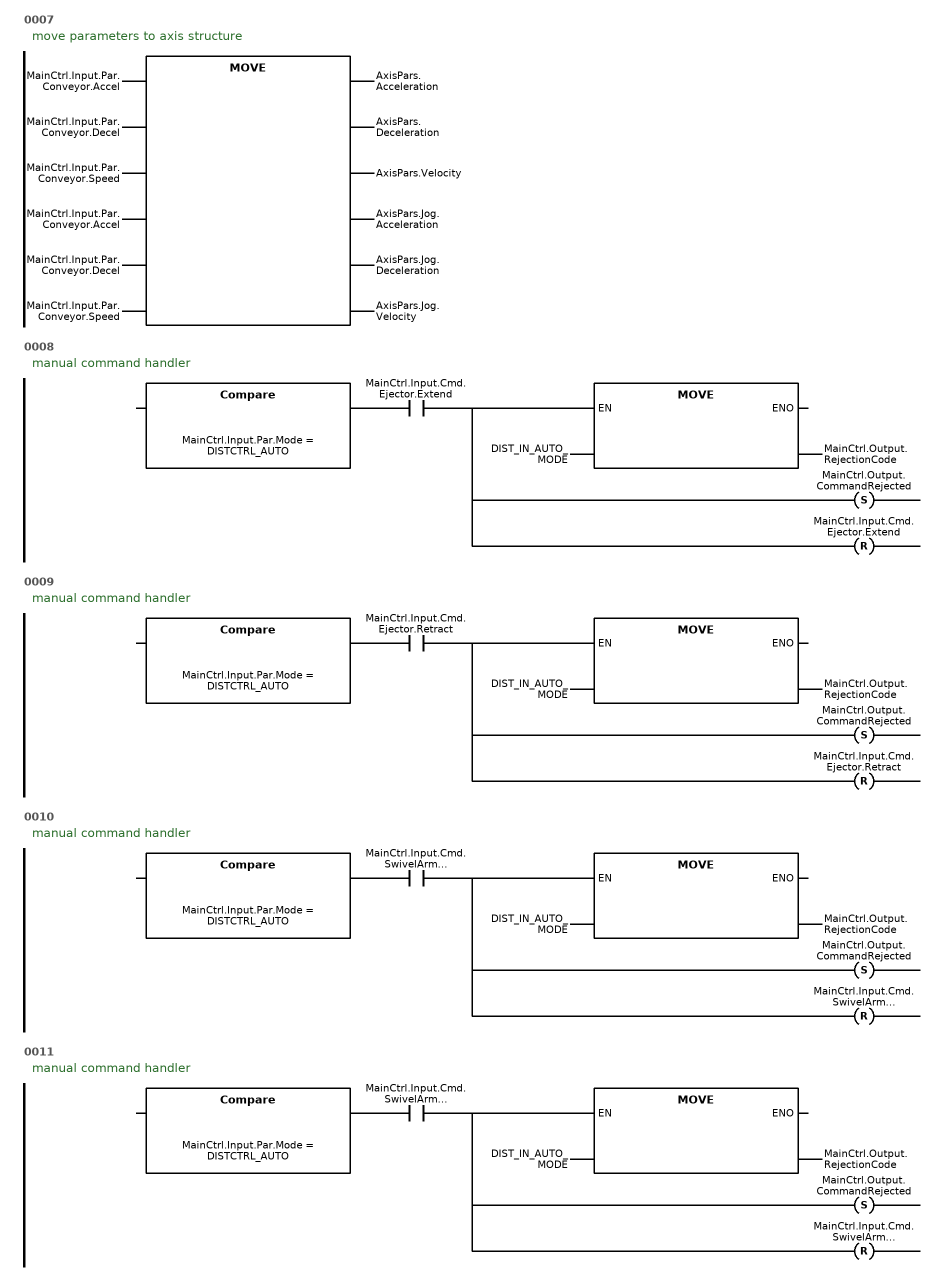
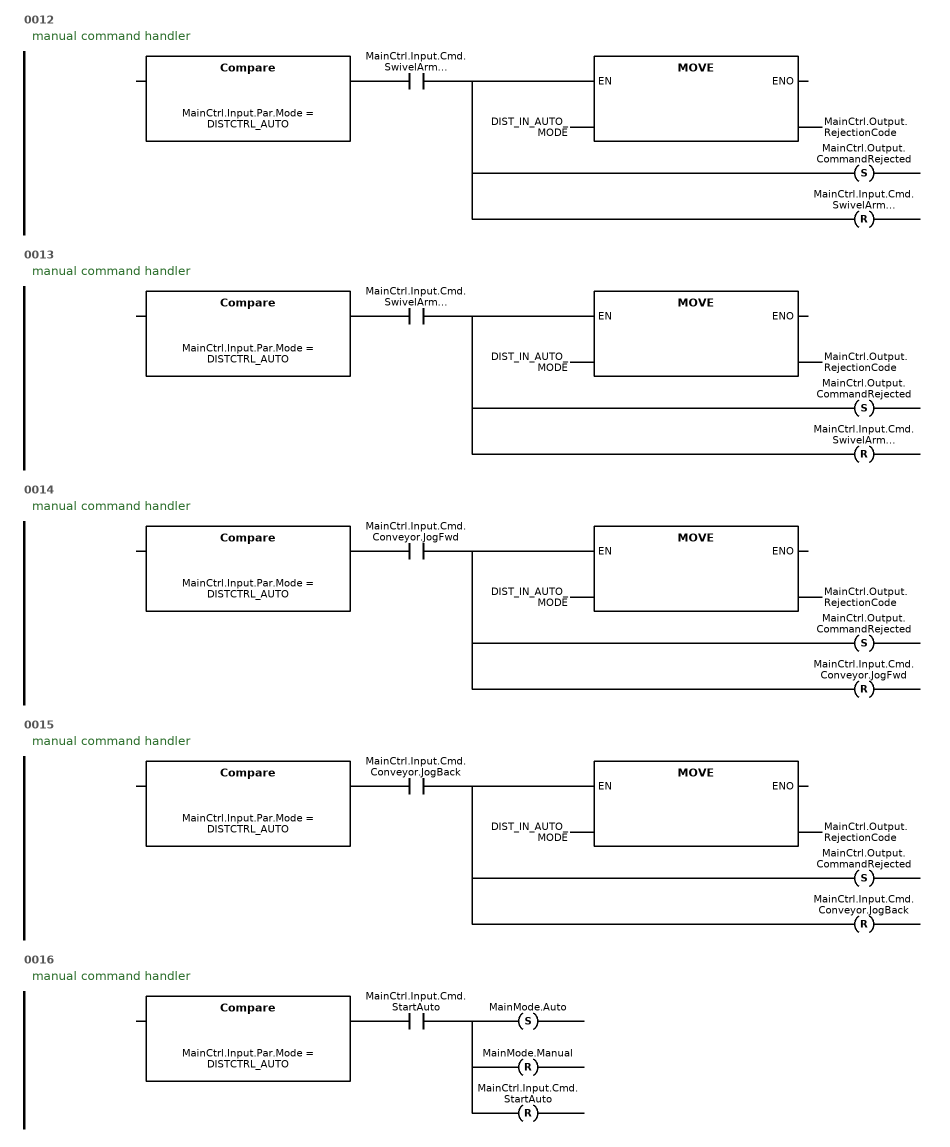
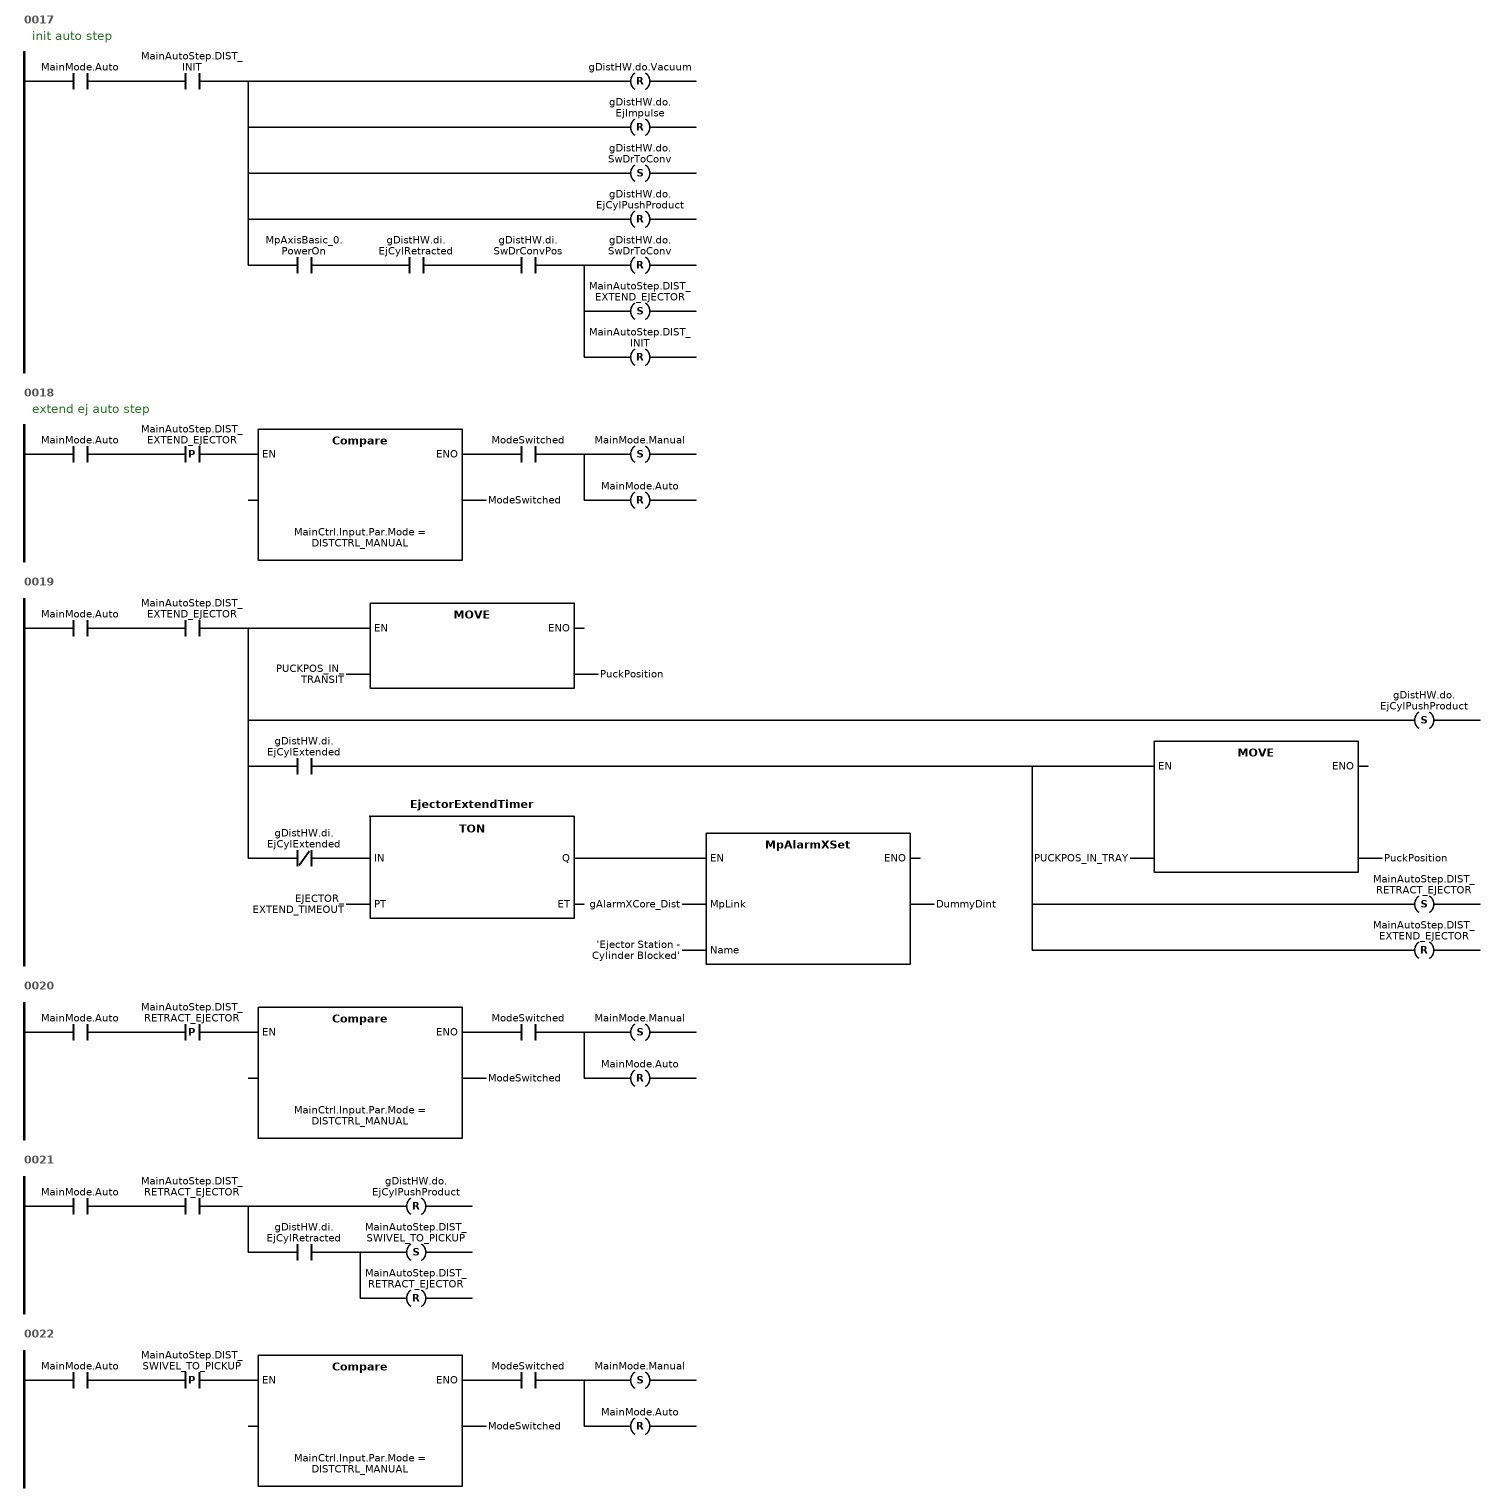
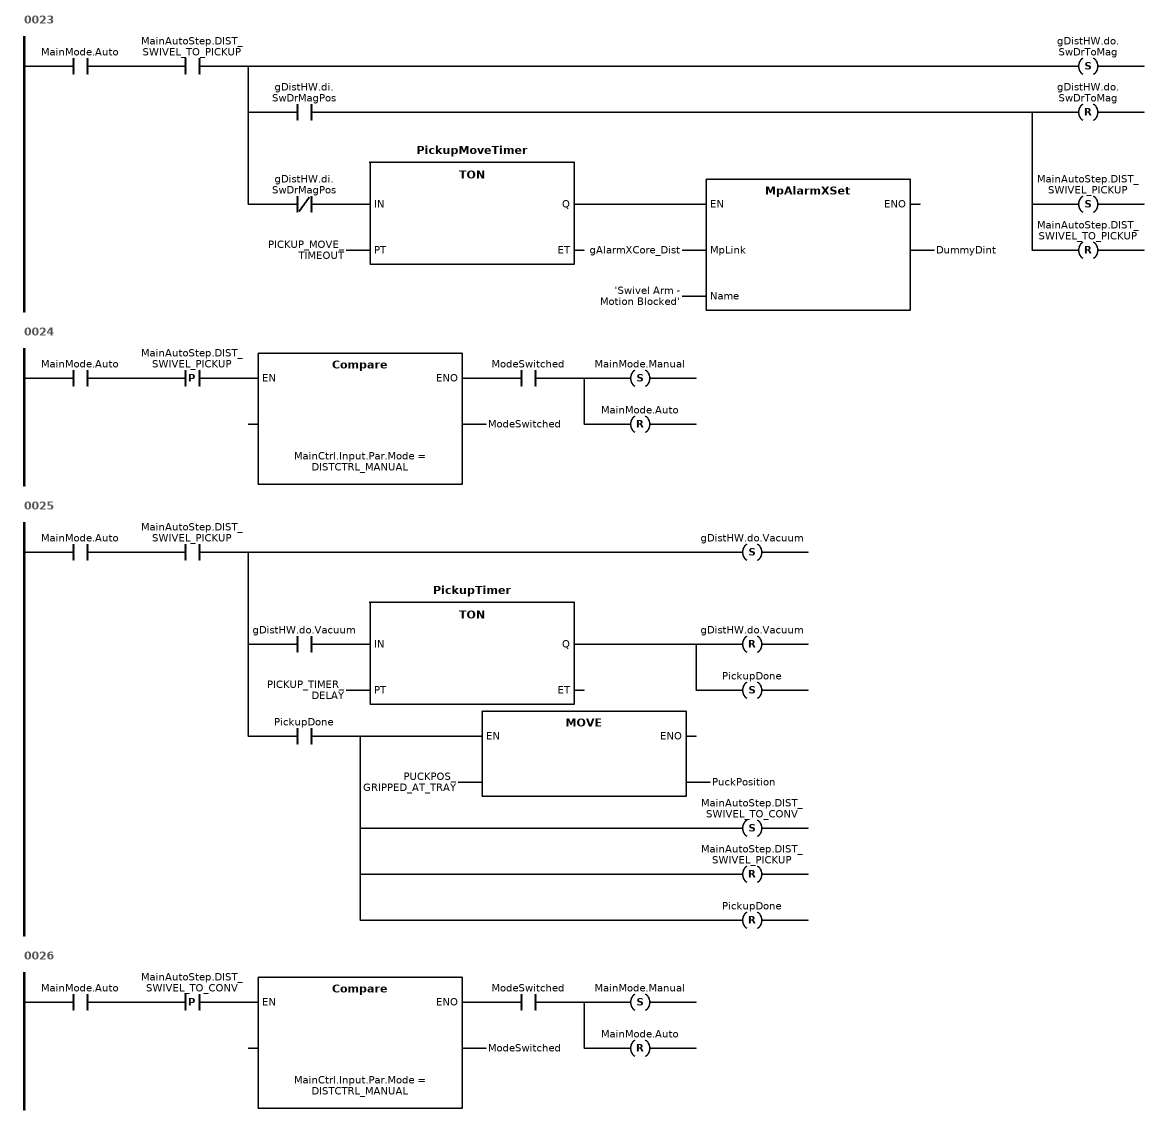
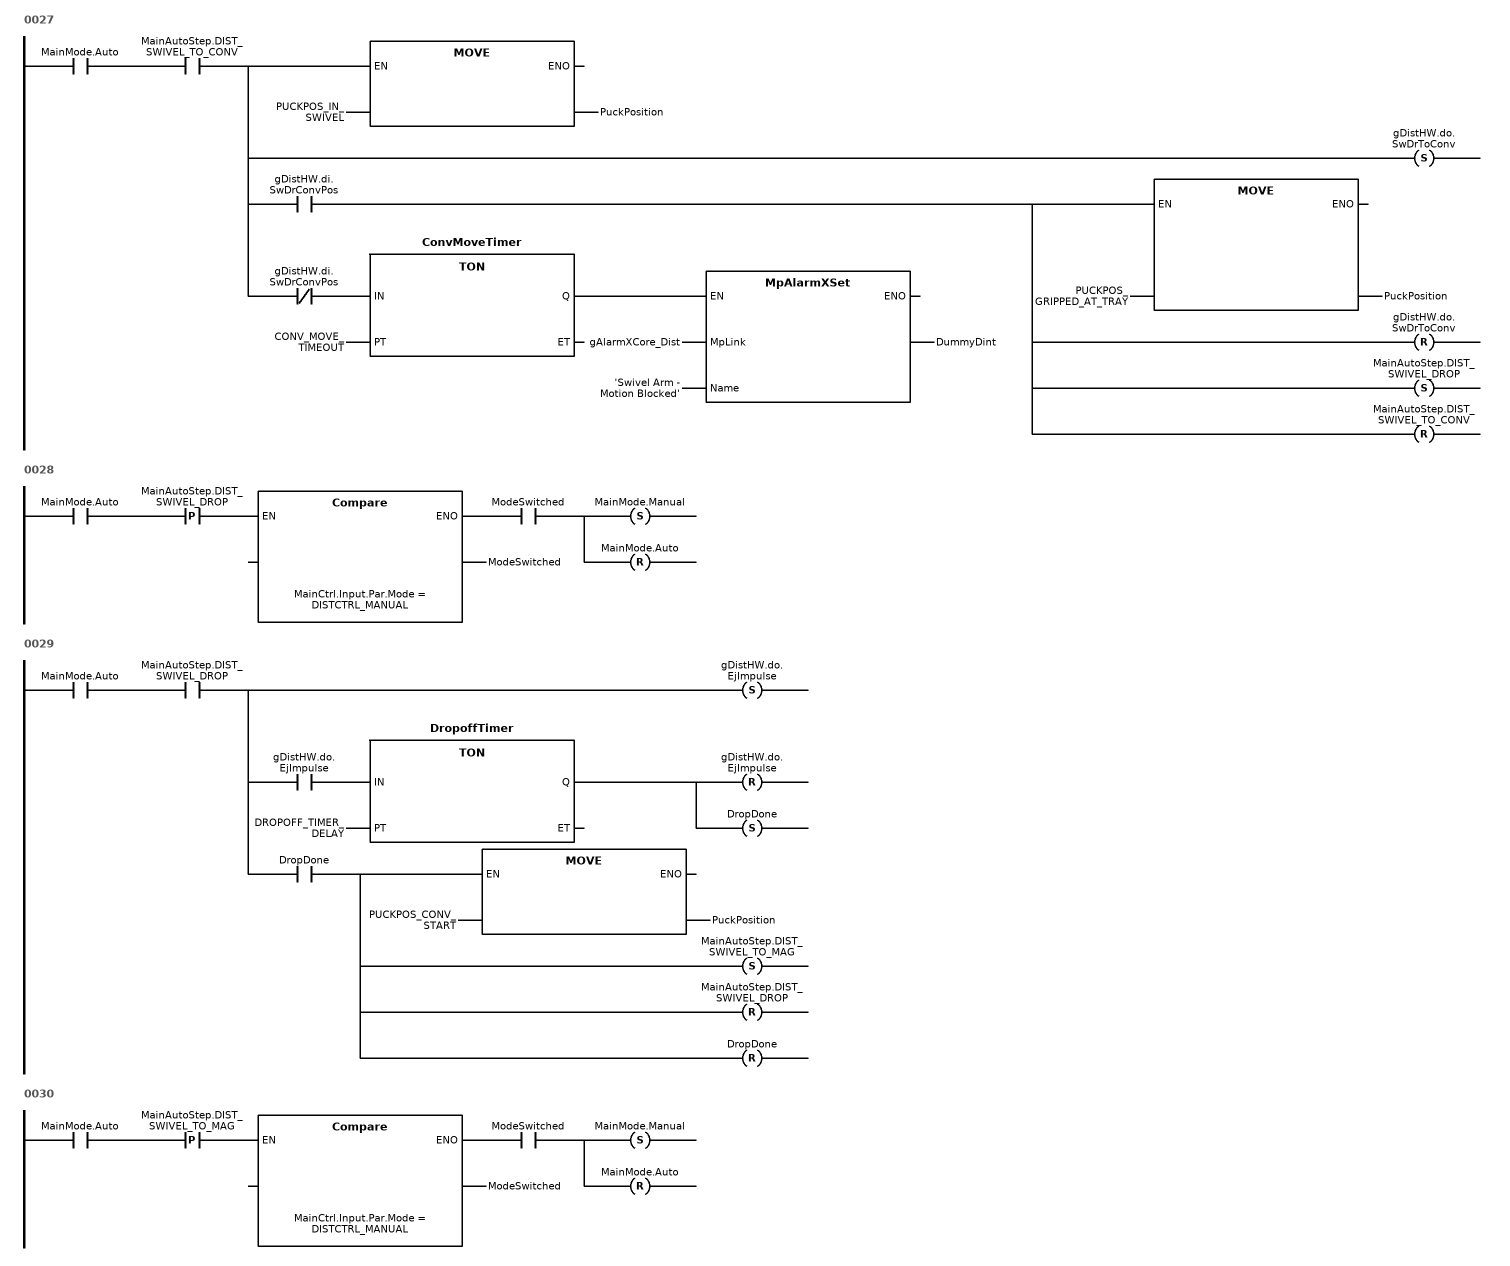
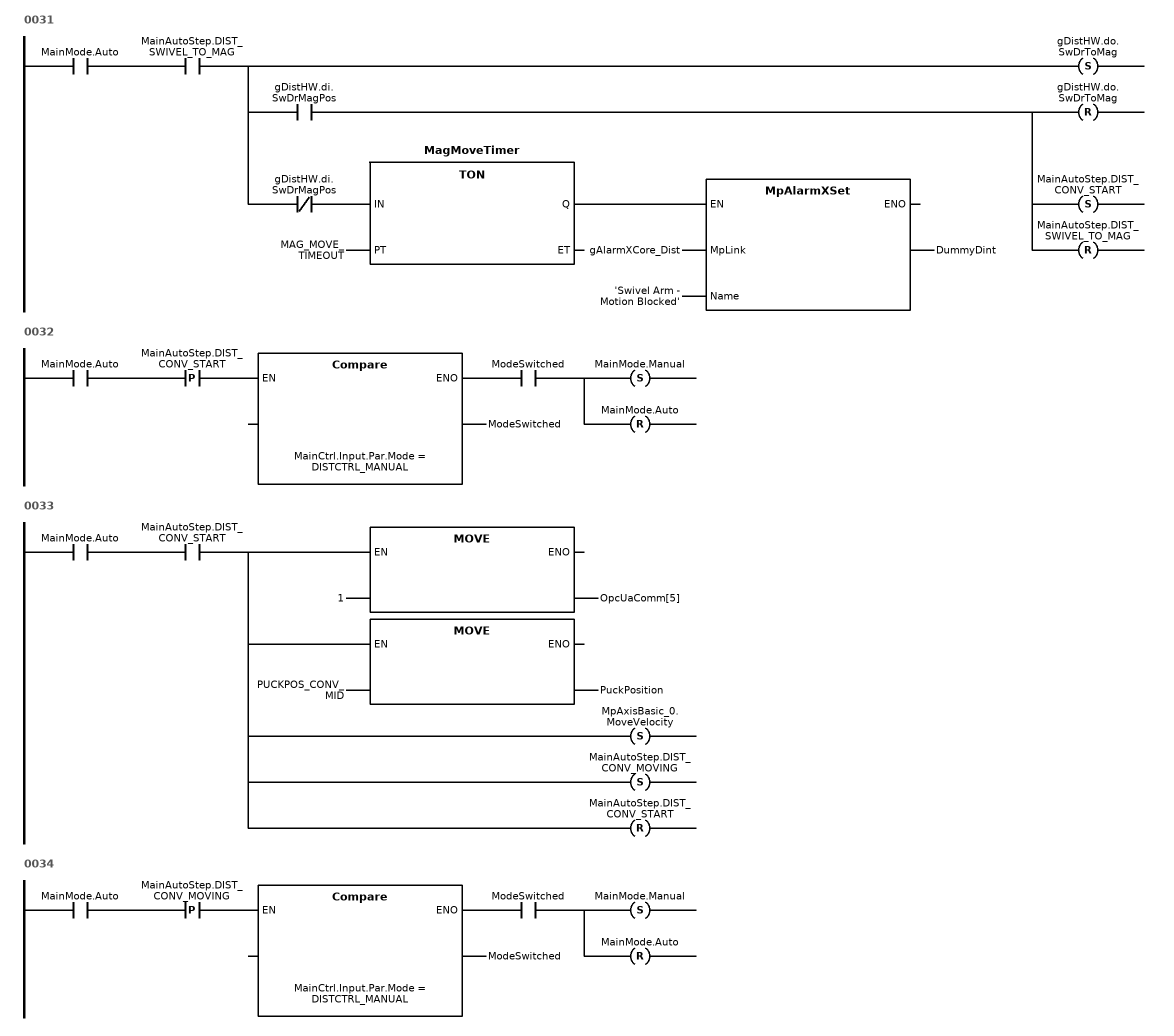
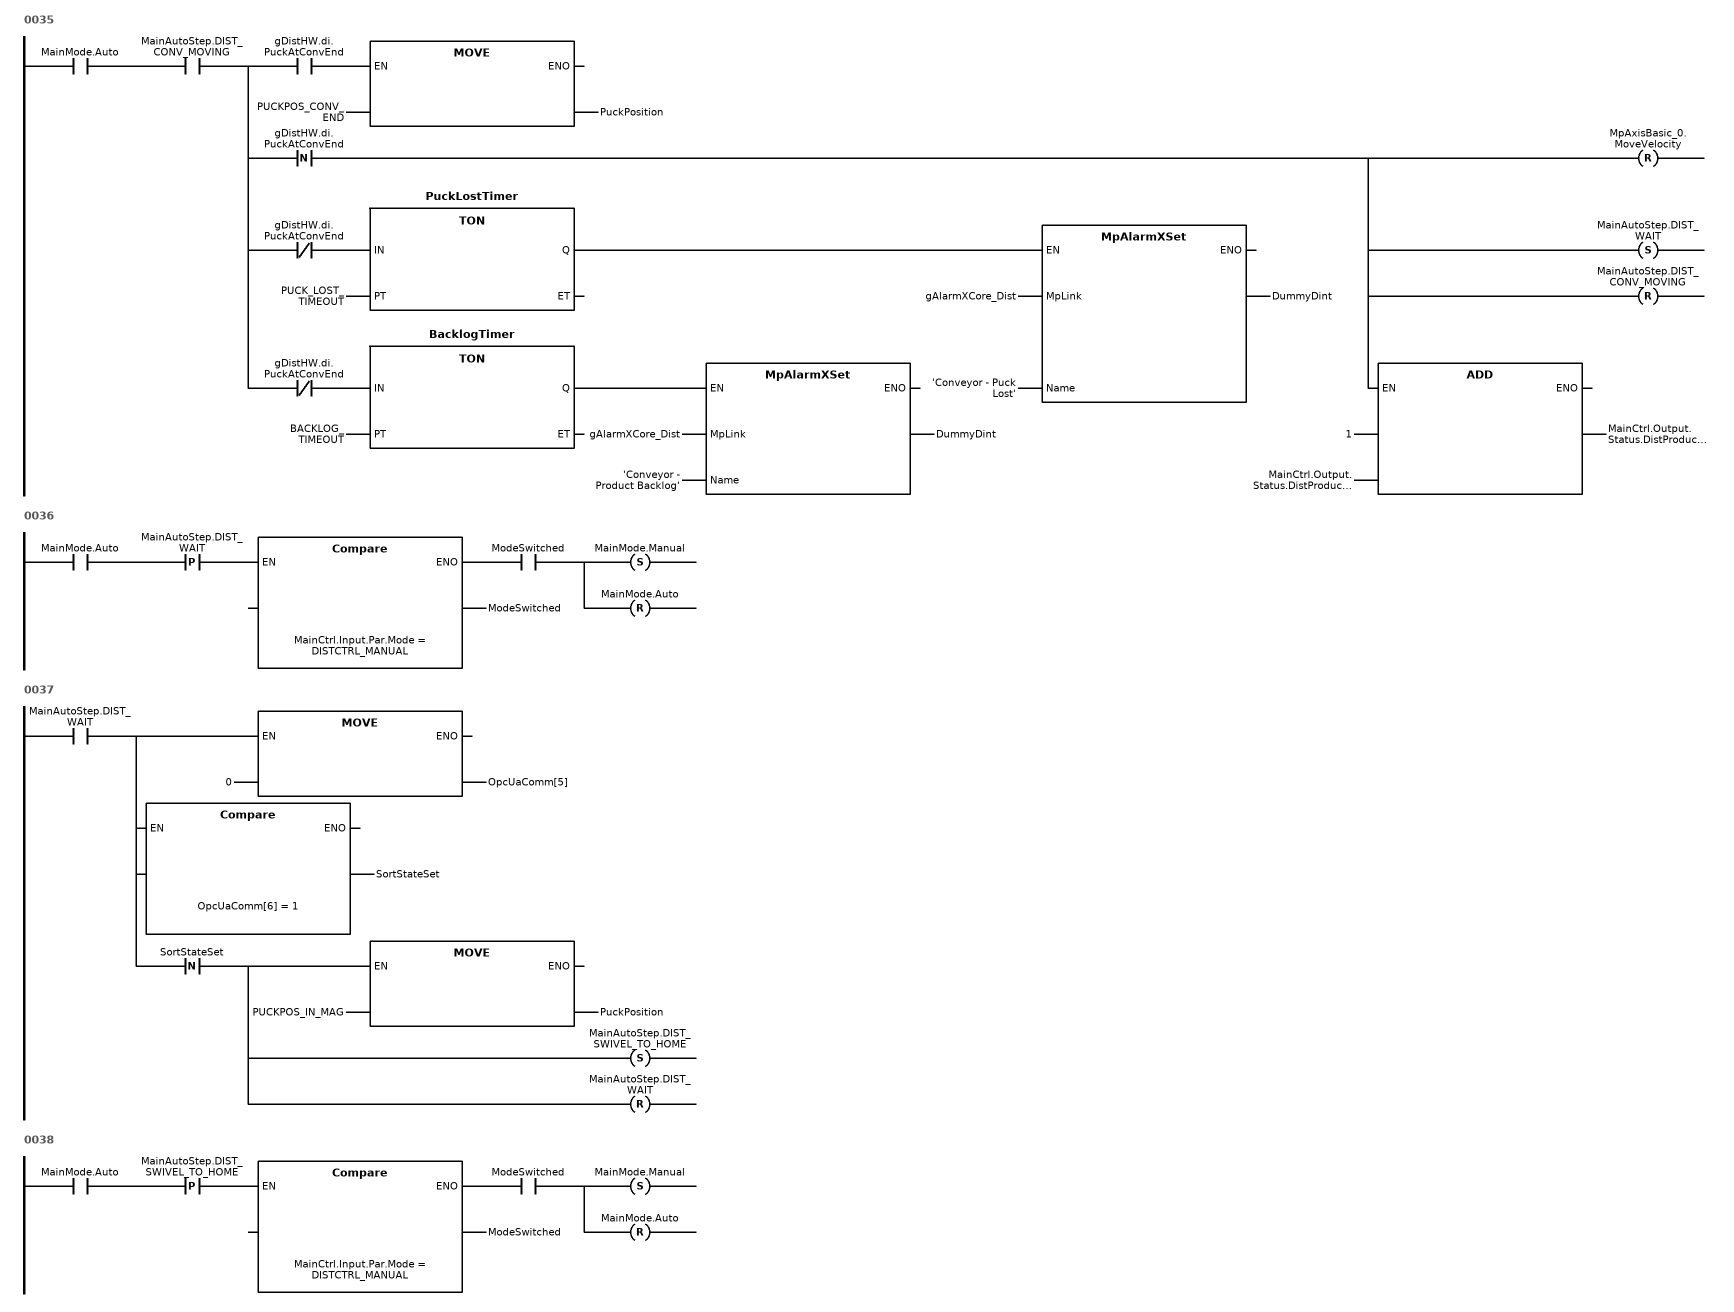
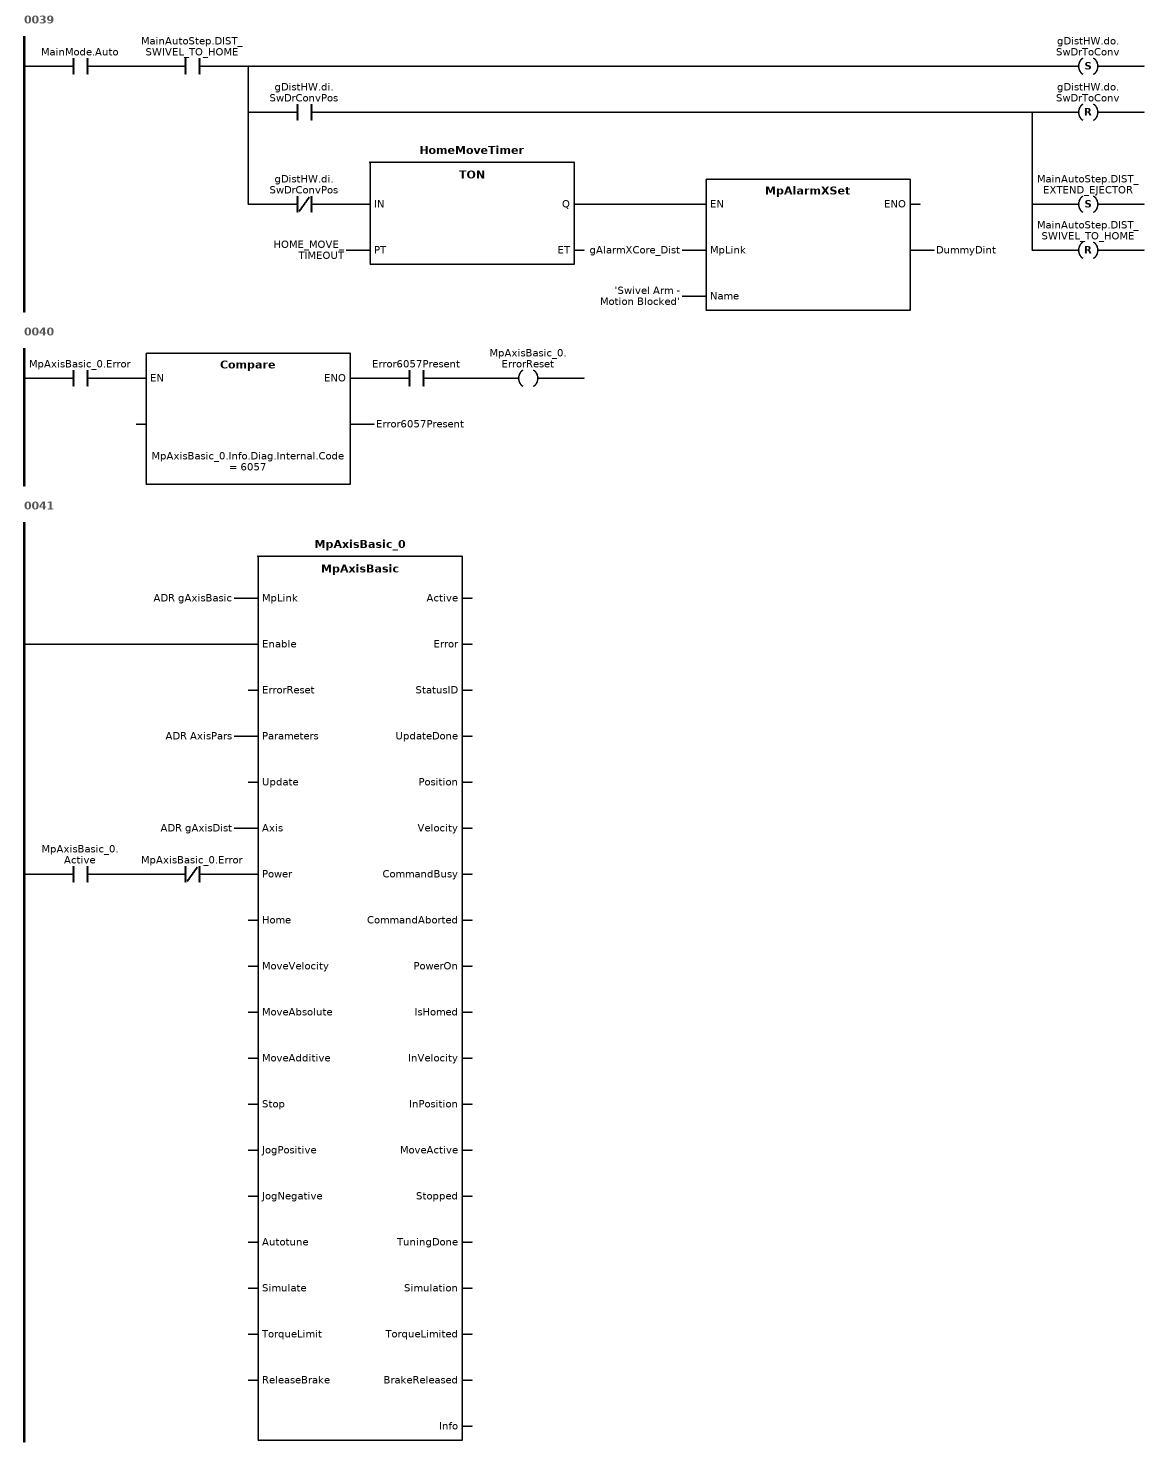
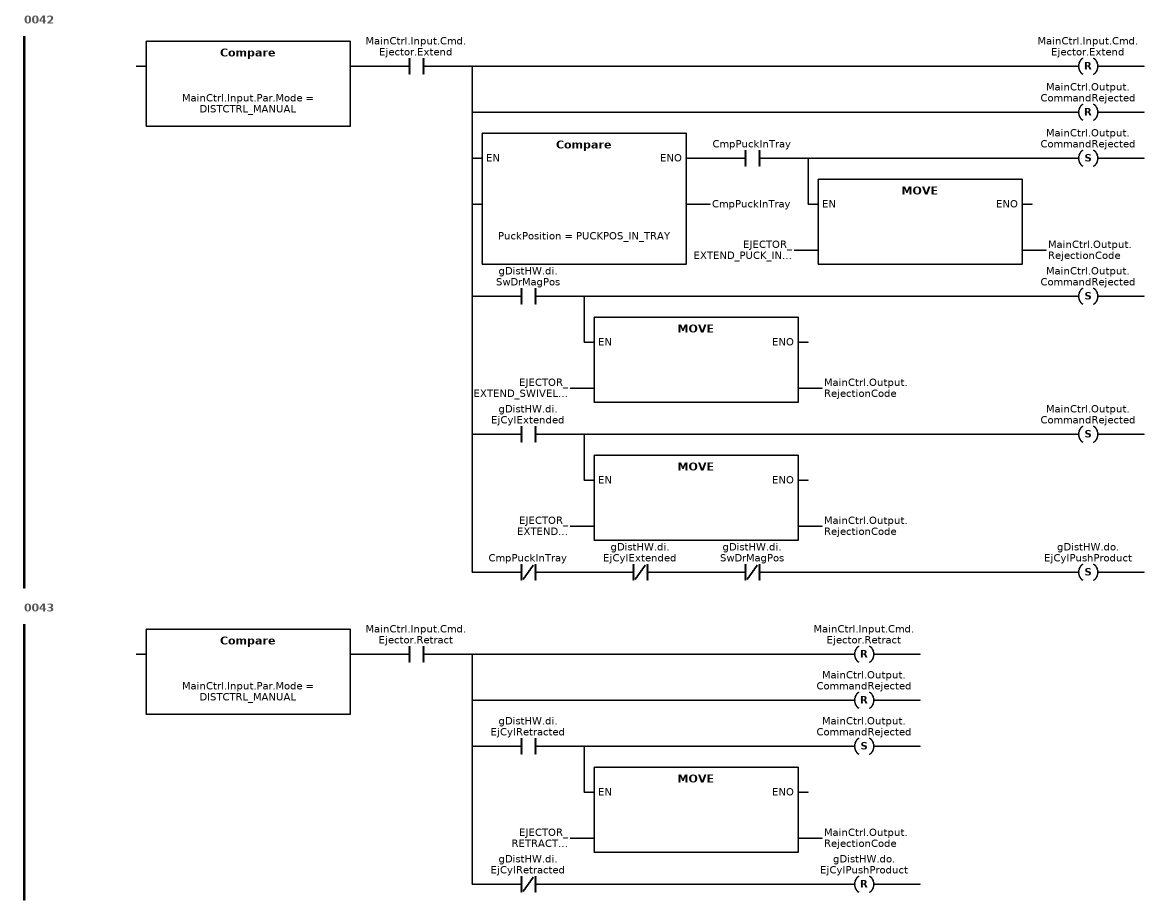
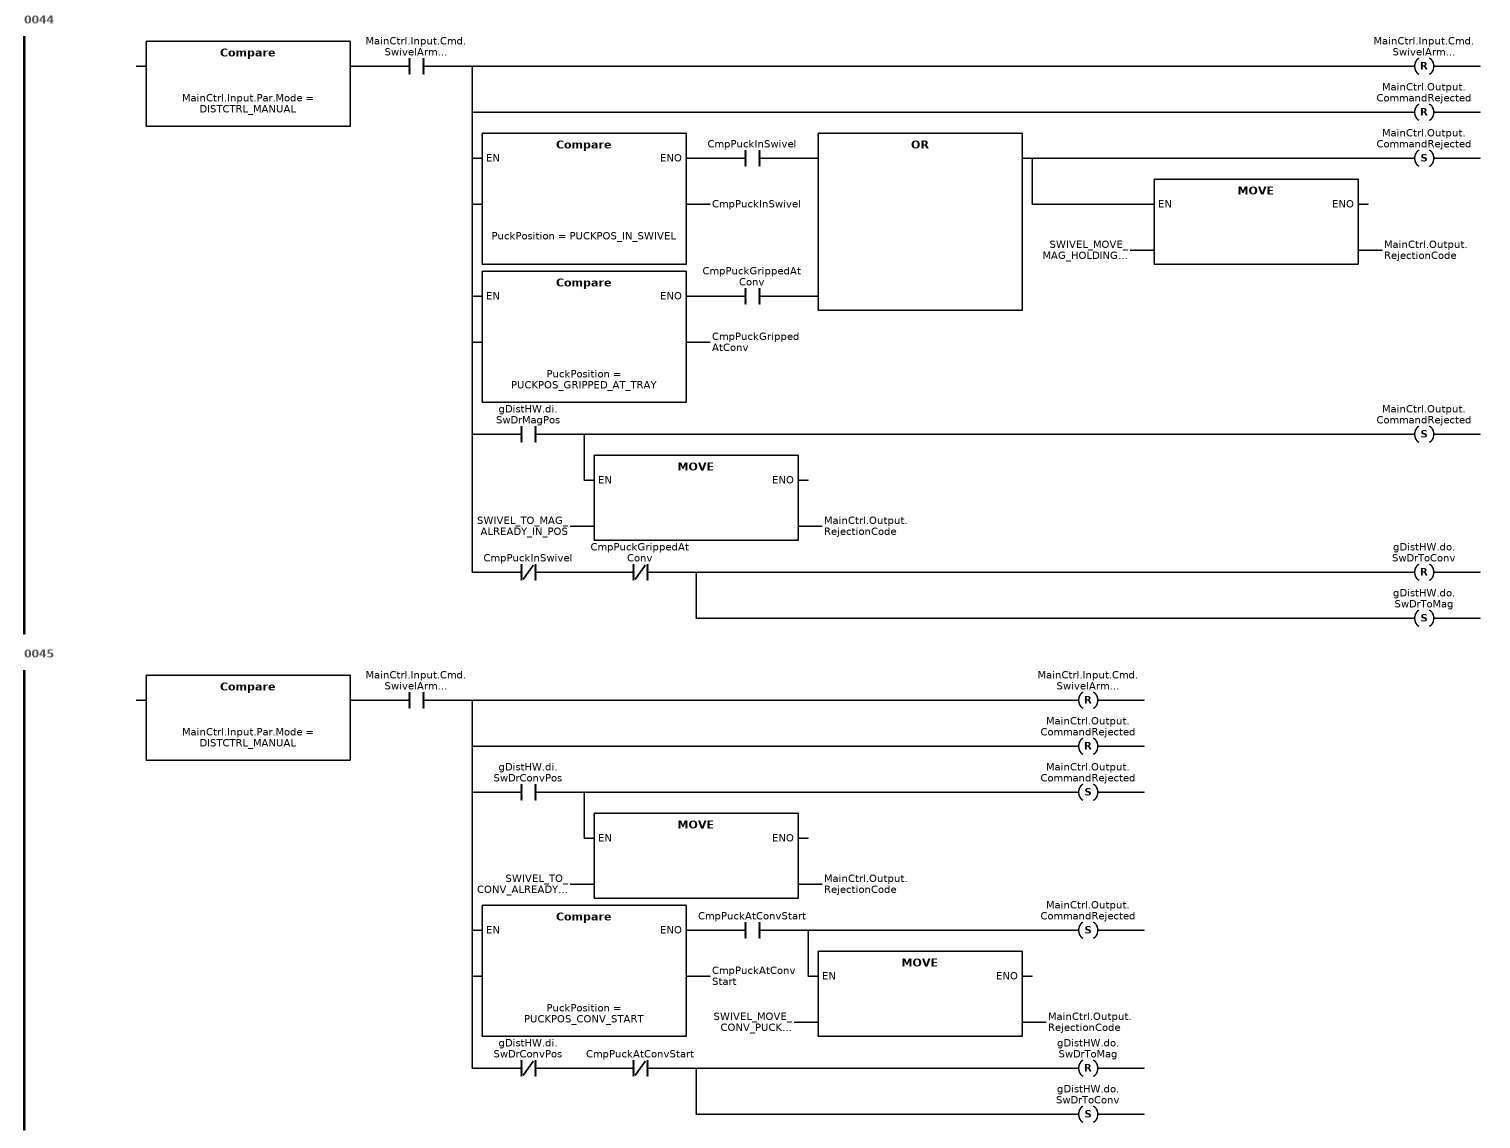
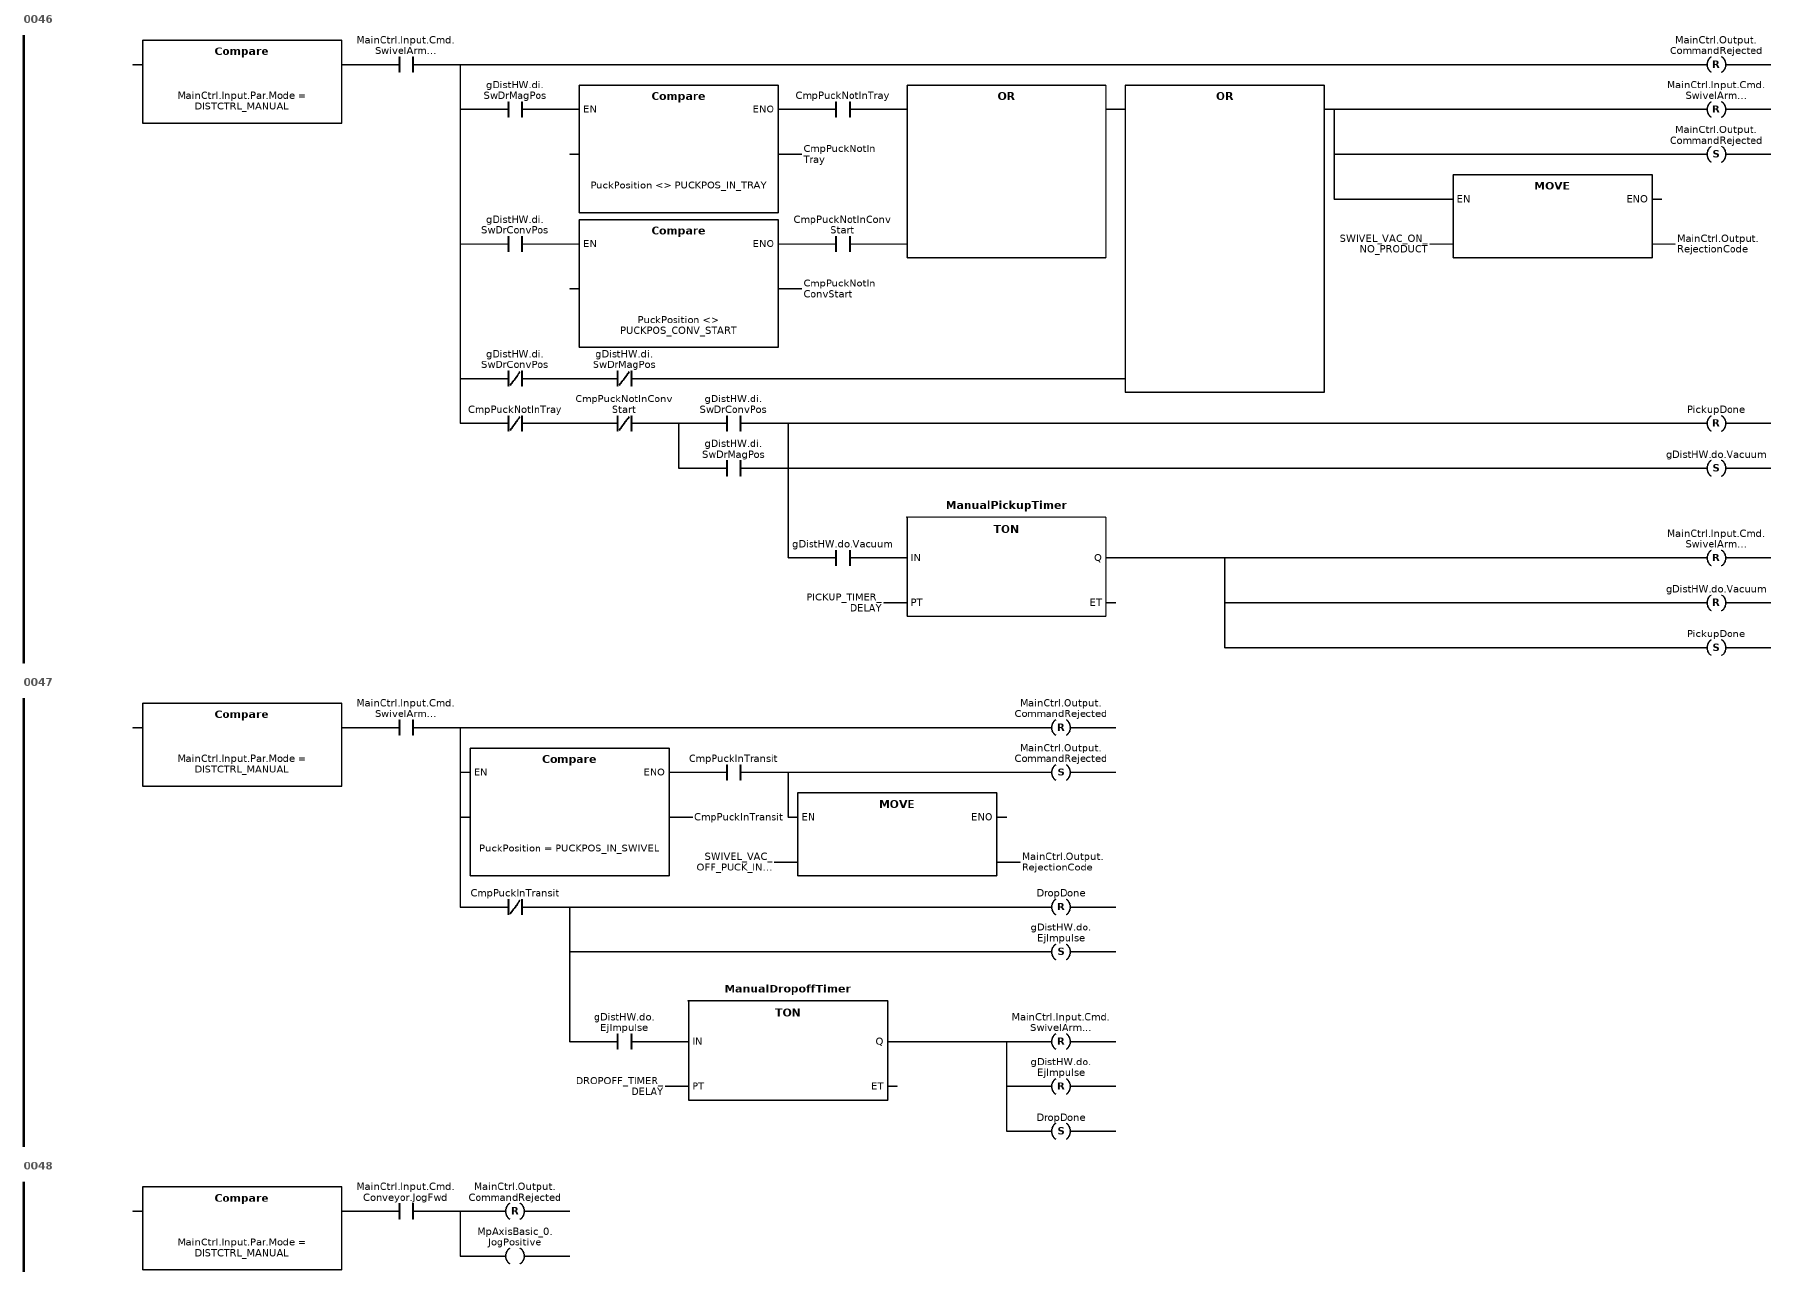
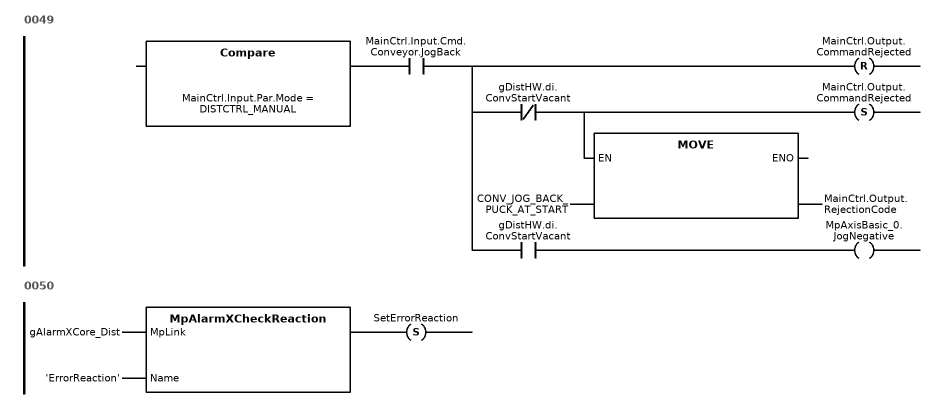
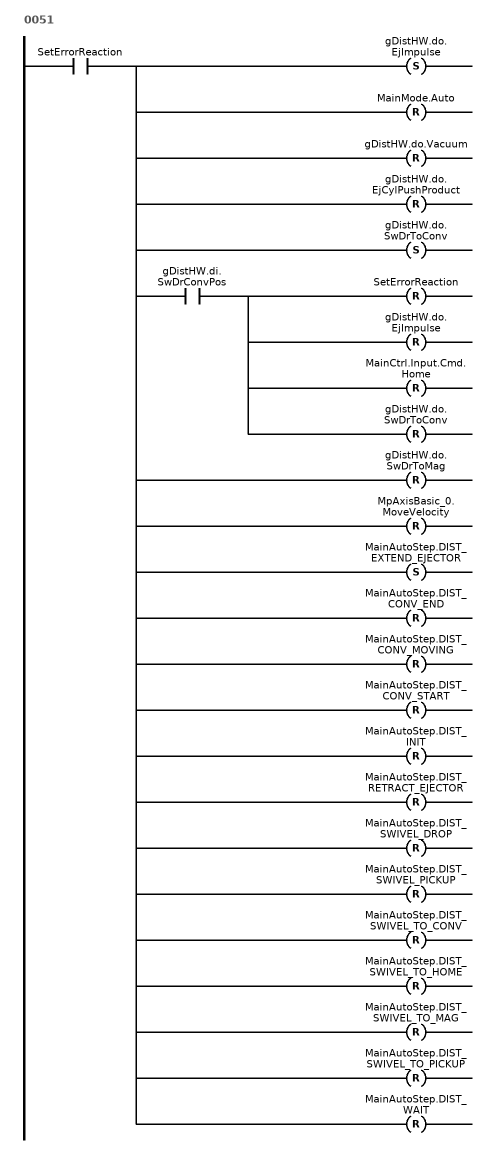
Ladder, written as Structured Text:
```iecst
(*********************************************************************************
 * Copyright:
 * Author:
 * Created:   	March 8, 2019/12:31 PM
 * Description:
 *********************************************************************************)

PROGRAM _CYCLIC
VAR
    _e1 : R_TRIG;
    _p2 : BOOL;
    _p3 : BOOL;
    _p4 : BOOL;
    _p5 : BOOL;
    _t6 : DINT;
    _e7 : R_TRIG;
    _p8 : BOOL;
    _p9 : BOOL;
    _p10 : BOOL;
    _p11 : BOOL;
    _p12 : BOOL;
    _p13 : BOOL;
    _p14 : BOOL;
    _p15 : BOOL;
    _p16 : BOOL;
    _p17 : BOOL;
    _e18 : R_TRIG;
    _p19 : BOOL;
    _p20 : BOOL;
    _e21 : R_TRIG;
    _p22 : BOOL;
    _p23 : BOOL;
    _e24 : R_TRIG;
    _p25 : BOOL;
    _p26 : BOOL;
    _p27 : BOOL;
    _e28 : R_TRIG;
    _p29 : BOOL;
    _p30 : BOOL;
    _e31 : R_TRIG;
    _p32 : BOOL;
    _p33 : BOOL;
    _p34 : BOOL;
    _e35 : R_TRIG;
    _p36 : BOOL;
    _p37 : BOOL;
    _e38 : R_TRIG;
    _p39 : BOOL;
    _p40 : BOOL;
    _p41 : BOOL;
    _e42 : R_TRIG;
    _p43 : BOOL;
    _p44 : BOOL;
    _e45 : R_TRIG;
    _p46 : BOOL;
    _e47 : F_TRIG;
    _p48 : BOOL;
    _p49 : BOOL;
    _e50 : R_TRIG;
    _p51 : BOOL;
    _e52 : F_TRIG;
    _p53 : BOOL;
    _e54 : R_TRIG;
    _p55 : BOOL;
    _p56 : BOOL;
    _p57 : BOOL;
    _p58 : BOOL;
    _p59 : BOOL;
    _p60 : BOOL;
    _t61 : BOOL;
    _p62 : BOOL;
    _p63 : BOOL;
    _p64 : BOOL;
    _p65 : BOOL;
    _t66 : BOOL;
    _p67 : BOOL;
    _p68 : BOOL;
    _p69 : BOOL;
    _p70 : BOOL;
    _p71 : BOOL;
    _p72 : BOOL;
    _p73 : BOOL;
    _p74 : BOOL;
END_VAR
(* Network 1: Handle OpcUa manual/automatic selection *)
IF (OpcUaComm[0] = 1) THEN
    MainCtrl.Input.Par.Mode := DISTCTRL_AUTO;
    SorterInControl := OpcUaComm[1] = 1;
END_IF;
IF (OpcUaComm[0] = 1) AND SorterInControl THEN StartAutoRequested := OpcUaComm[2] = 1; END_IF;
_e1(CLK := StartAutoRequested);
IF (OpcUaComm[0] = 1) AND SorterInControl AND _e1.Q THEN
    MainMode.Auto := TRUE;
    MainMode.Manual := FALSE;
END_IF;

(* Network 2: Reset auto mode over opc ua *)
_p2 := MainCtrl.Input.Cmd.StopAuto;
IF MainCtrl.Input.Cmd.StopAuto THEN MainCtrl.Input.Cmd.StopAuto := FALSE; END_IF;
IF _p2 THEN OpcUaComm[0] := 0; END_IF;

(* Network 3: Set manual mode based on opc ua *)
IF (OpcUaComm[0] = 0) THEN
    MainCtrl.Input.Par.Mode := DISTCTRL_MANUAL;
    MainMode.Auto := FALSE;
    MainMode.Manual := TRUE;
END_IF;

(* Network 4: handle homing commands *)
IF MainCtrl.Input.Cmd.Home THEN
    gDistHW.do.EjImpulse := TRUE;
    MainMode.Auto := FALSE;
    gDistHW.do.Vacuum := FALSE;
    gDistHW.do.EjCylPushProduct := FALSE;
    gDistHW.do.SwDrToConv := TRUE;
END_IF;
_p3 := MainCtrl.Input.Cmd.Home AND gDistHW.di.SwDrConvPos;
IF _p3 THEN gDistHW.do.EjImpulse := FALSE; END_IF;
_p4 := MainCtrl.Input.Cmd.Home;
IF _p3 THEN
    MainCtrl.Input.Cmd.Home := FALSE;
    gDistHW.do.SwDrToConv := FALSE;
END_IF;
IF _p4 THEN
    gDistHW.do.SwDrToMag := FALSE;
    MpAxisBasic_0.MoveVelocity := FALSE;
    MainAutoStep.DIST_EXTEND_EJECTOR := TRUE;
    MainAutoStep.DIST_CONV_END := FALSE;
    MainAutoStep.DIST_CONV_MOVING := FALSE;
    MainAutoStep.DIST_CONV_START := FALSE;
    MainAutoStep.DIST_INIT := FALSE;
    MainAutoStep.DIST_RETRACT_EJECTOR := FALSE;
    MainAutoStep.DIST_SWIVEL_DROP := FALSE;
    MainAutoStep.DIST_SWIVEL_PICKUP := FALSE;
    MainAutoStep.DIST_SWIVEL_TO_CONV := FALSE;
    MainAutoStep.DIST_SWIVEL_TO_HOME := FALSE;
    MainAutoStep.DIST_SWIVEL_TO_MAG := FALSE;
    MainAutoStep.DIST_SWIVEL_TO_PICKUP := FALSE;
    MainAutoStep.DIST_WAIT := FALSE;
END_IF;

(* Network 5: Reset counter and timer *)
_p5 := MainCtrl.Input.Cmd.Reset;
IF _p5 THEN MainCtrl.Output.Status.AutoRunTime := T#0s; END_IF;
_t6 := MainCtrl.Output.Status.AutoRunTime;
IF _p5 THEN
    MainCtrl.Input.Cmd.Reset := FALSE;
    MainCtrl.Output.Status.DistProductCount := 0;
END_IF;

(* Network 6: Set opcua communication if auto selected *)
AutoSelected := MainCtrl.Input.Par.Mode = DISTCTRL_AUTO;
_e7(CLK := AutoSelected);
IF _e7.Q THEN OpcUaComm[0] := 1; END_IF;

(* Network 7: move parameters to axis structure *)
AxisPars.Acceleration := MainCtrl.Input.Par.Conveyor.Accel;
AxisPars.Deceleration := MainCtrl.Input.Par.Conveyor.Decel;
AxisPars.Velocity := MainCtrl.Input.Par.Conveyor.Speed;
AxisPars.Jog.Acceleration := MainCtrl.Input.Par.Conveyor.Accel;
AxisPars.Jog.Deceleration := MainCtrl.Input.Par.Conveyor.Decel;
AxisPars.Jog.Velocity := MainCtrl.Input.Par.Conveyor.Speed;

(* Network 8: manual command handler *)
_p8 := (MainCtrl.Input.Par.Mode = DISTCTRL_AUTO) AND MainCtrl.Input.Cmd.Ejector.Extend;
IF _p8 THEN
    MainCtrl.Output.RejectionCode := DIST_IN_AUTO_MODE;
    MainCtrl.Output.CommandRejected := TRUE;
    MainCtrl.Input.Cmd.Ejector.Extend := FALSE;
END_IF;

(* Network 9: manual command handler *)
_p9 := (MainCtrl.Input.Par.Mode = DISTCTRL_AUTO) AND MainCtrl.Input.Cmd.Ejector.Retract;
IF _p9 THEN
    MainCtrl.Output.RejectionCode := DIST_IN_AUTO_MODE;
    MainCtrl.Output.CommandRejected := TRUE;
    MainCtrl.Input.Cmd.Ejector.Retract := FALSE;
END_IF;

(* Network 10: manual command handler *)
_p10 := (MainCtrl.Input.Par.Mode = DISTCTRL_AUTO) AND MainCtrl.Input.Cmd.SwivelArm.MoveToConveyor;
IF _p10 THEN
    MainCtrl.Output.RejectionCode := DIST_IN_AUTO_MODE;
    MainCtrl.Output.CommandRejected := TRUE;
    MainCtrl.Input.Cmd.SwivelArm.MoveToConveyor := FALSE;
END_IF;

(* Network 11: manual command handler *)
_p11 := (MainCtrl.Input.Par.Mode = DISTCTRL_AUTO) AND MainCtrl.Input.Cmd.SwivelArm.MoveToMagazine;
IF _p11 THEN
    MainCtrl.Output.RejectionCode := DIST_IN_AUTO_MODE;
    MainCtrl.Output.CommandRejected := TRUE;
    MainCtrl.Input.Cmd.SwivelArm.MoveToMagazine := FALSE;
END_IF;

(* Network 12: manual command handler *)
_p12 := (MainCtrl.Input.Par.Mode = DISTCTRL_AUTO) AND MainCtrl.Input.Cmd.SwivelArm.VacuumOnImpulse;
IF _p12 THEN
    MainCtrl.Output.RejectionCode := DIST_IN_AUTO_MODE;
    MainCtrl.Output.CommandRejected := TRUE;
    MainCtrl.Input.Cmd.SwivelArm.VacuumOnImpulse := FALSE;
END_IF;

(* Network 13: manual command handler *)
_p13 := (MainCtrl.Input.Par.Mode = DISTCTRL_AUTO) AND MainCtrl.Input.Cmd.SwivelArm.VacuumOffImpulse;
IF _p13 THEN
    MainCtrl.Output.RejectionCode := DIST_IN_AUTO_MODE;
    MainCtrl.Output.CommandRejected := TRUE;
    MainCtrl.Input.Cmd.SwivelArm.VacuumOffImpulse := FALSE;
END_IF;

(* Network 14: manual command handler *)
_p14 := (MainCtrl.Input.Par.Mode = DISTCTRL_AUTO) AND MainCtrl.Input.Cmd.Conveyor.JogFwd;
IF _p14 THEN
    MainCtrl.Output.RejectionCode := DIST_IN_AUTO_MODE;
    MainCtrl.Output.CommandRejected := TRUE;
    MainCtrl.Input.Cmd.Conveyor.JogFwd := FALSE;
END_IF;

(* Network 15: manual command handler *)
_p15 := (MainCtrl.Input.Par.Mode = DISTCTRL_AUTO) AND MainCtrl.Input.Cmd.Conveyor.JogBack;
IF _p15 THEN
    MainCtrl.Output.RejectionCode := DIST_IN_AUTO_MODE;
    MainCtrl.Output.CommandRejected := TRUE;
    MainCtrl.Input.Cmd.Conveyor.JogBack := FALSE;
END_IF;

(* Network 16: manual command handler *)
_p16 := (MainCtrl.Input.Par.Mode = DISTCTRL_AUTO) AND MainCtrl.Input.Cmd.StartAuto;
IF _p16 THEN
    MainMode.Auto := TRUE;
    MainMode.Manual := FALSE;
    MainCtrl.Input.Cmd.StartAuto := FALSE;
END_IF;

(* Network 17: init auto step *)
IF MainMode.Auto AND MainAutoStep.DIST_INIT THEN
    gDistHW.do.Vacuum := FALSE;
    gDistHW.do.EjImpulse := FALSE;
    gDistHW.do.SwDrToConv := TRUE;
    gDistHW.do.EjCylPushProduct := FALSE;
END_IF;
_p17 := MainMode.Auto AND MainAutoStep.DIST_INIT AND MpAxisBasic_0.PowerOn AND gDistHW.di.EjCylRetracted AND gDistHW.di.SwDrConvPos;
IF _p17 THEN
    gDistHW.do.SwDrToConv := FALSE;
    MainAutoStep.DIST_EXTEND_EJECTOR := TRUE;
    MainAutoStep.DIST_INIT := FALSE;
END_IF;

(* Network 18: extend ej auto step *)
_e18(CLK := MainAutoStep.DIST_EXTEND_EJECTOR);
IF MainMode.Auto AND _e18.Q THEN ModeSwitched := MainCtrl.Input.Par.Mode = DISTCTRL_MANUAL; END_IF;
_p19 := MainMode.Auto AND _e18.Q AND ModeSwitched;
IF MainMode.Auto AND _e18.Q AND ModeSwitched THEN MainMode.Manual := TRUE; END_IF;
IF _p19 THEN MainMode.Auto := FALSE; END_IF;

(* Network 19 *)
_p20 := MainMode.Auto AND MainAutoStep.DIST_EXTEND_EJECTOR;
IF _p20 THEN
    PuckPosition := PUCKPOS_IN_TRANSIT;
    gDistHW.do.EjCylPushProduct := TRUE;
END_IF;
EjectorExtendTimer(IN := _p20 AND NOT gDistHW.di.EjCylExtended, PT := EJECTOR_EXTEND_TIMEOUT);
IF _p20 AND gDistHW.di.EjCylExtended THEN PuckPosition := PUCKPOS_IN_TRAY; END_IF;
IF EjectorExtendTimer.Q THEN
    DummyDint := MpAlarmXSet(MpLink := gAlarmXCore_Dist, Name := 'Ejector Station - Cylinder Blocked');
END_IF;
IF _p20 AND gDistHW.di.EjCylExtended THEN
    MainAutoStep.DIST_RETRACT_EJECTOR := TRUE;
    MainAutoStep.DIST_EXTEND_EJECTOR := FALSE;
END_IF;

(* Network 20 *)
_e21(CLK := MainAutoStep.DIST_RETRACT_EJECTOR);
IF MainMode.Auto AND _e21.Q THEN ModeSwitched := MainCtrl.Input.Par.Mode = DISTCTRL_MANUAL; END_IF;
_p22 := MainMode.Auto AND _e21.Q AND ModeSwitched;
IF MainMode.Auto AND _e21.Q AND ModeSwitched THEN MainMode.Manual := TRUE; END_IF;
IF _p22 THEN MainMode.Auto := FALSE; END_IF;

(* Network 21 *)
_p23 := MainMode.Auto AND MainAutoStep.DIST_RETRACT_EJECTOR;
IF _p23 THEN gDistHW.do.EjCylPushProduct := FALSE; END_IF;
IF _p23 AND gDistHW.di.EjCylRetracted THEN
    MainAutoStep.DIST_SWIVEL_TO_PICKUP := TRUE;
    MainAutoStep.DIST_RETRACT_EJECTOR := FALSE;
END_IF;

(* Network 22 *)
_e24(CLK := MainAutoStep.DIST_SWIVEL_TO_PICKUP);
IF MainMode.Auto AND _e24.Q THEN ModeSwitched := MainCtrl.Input.Par.Mode = DISTCTRL_MANUAL; END_IF;
_p25 := MainMode.Auto AND _e24.Q AND ModeSwitched;
IF MainMode.Auto AND _e24.Q AND ModeSwitched THEN MainMode.Manual := TRUE; END_IF;
IF _p25 THEN MainMode.Auto := FALSE; END_IF;

(* Network 23 *)
_p26 := MainMode.Auto AND MainAutoStep.DIST_SWIVEL_TO_PICKUP;
IF _p26 THEN gDistHW.do.SwDrToMag := TRUE; END_IF;
_p27 := _p26 AND gDistHW.di.SwDrMagPos;
IF _p26 AND gDistHW.di.SwDrMagPos THEN gDistHW.do.SwDrToMag := FALSE; END_IF;
PickupMoveTimer(IN := _p26 AND NOT gDistHW.di.SwDrMagPos, PT := PICKUP_MOVE_TIMEOUT);
IF _p27 THEN MainAutoStep.DIST_SWIVEL_PICKUP := TRUE; END_IF;
IF PickupMoveTimer.Q THEN
    DummyDint := MpAlarmXSet(MpLink := gAlarmXCore_Dist, Name := 'Swivel Arm - Motion Blocked');
END_IF;
IF _p27 THEN MainAutoStep.DIST_SWIVEL_TO_PICKUP := FALSE; END_IF;

(* Network 24 *)
_e28(CLK := MainAutoStep.DIST_SWIVEL_PICKUP);
IF MainMode.Auto AND _e28.Q THEN ModeSwitched := MainCtrl.Input.Par.Mode = DISTCTRL_MANUAL; END_IF;
_p29 := MainMode.Auto AND _e28.Q AND ModeSwitched;
IF MainMode.Auto AND _e28.Q AND ModeSwitched THEN MainMode.Manual := TRUE; END_IF;
IF _p29 THEN MainMode.Auto := FALSE; END_IF;

(* Network 25 *)
_p30 := MainMode.Auto AND MainAutoStep.DIST_SWIVEL_PICKUP;
IF _p30 THEN gDistHW.do.Vacuum := TRUE; END_IF;
PickupTimer(IN := _p30 AND gDistHW.do.Vacuum, PT := PICKUP_TIMER_DELAY);
IF PickupTimer.Q THEN
    gDistHW.do.Vacuum := FALSE;
    PickupDone := TRUE;
END_IF;
IF _p30 AND PickupDone THEN
    PuckPosition := PUCKPOS_GRIPPED_AT_TRAY;
    MainAutoStep.DIST_SWIVEL_TO_CONV := TRUE;
    MainAutoStep.DIST_SWIVEL_PICKUP := FALSE;
    PickupDone := FALSE;
END_IF;

(* Network 26 *)
_e31(CLK := MainAutoStep.DIST_SWIVEL_TO_CONV);
IF MainMode.Auto AND _e31.Q THEN ModeSwitched := MainCtrl.Input.Par.Mode = DISTCTRL_MANUAL; END_IF;
_p32 := MainMode.Auto AND _e31.Q AND ModeSwitched;
IF MainMode.Auto AND _e31.Q AND ModeSwitched THEN MainMode.Manual := TRUE; END_IF;
IF _p32 THEN MainMode.Auto := FALSE; END_IF;

(* Network 27 *)
_p33 := MainMode.Auto AND MainAutoStep.DIST_SWIVEL_TO_CONV;
IF _p33 THEN
    PuckPosition := PUCKPOS_IN_SWIVEL;
    gDistHW.do.SwDrToConv := TRUE;
END_IF;
ConvMoveTimer(IN := _p33 AND NOT gDistHW.di.SwDrConvPos, PT := CONV_MOVE_TIMEOUT);
IF _p33 AND gDistHW.di.SwDrConvPos THEN PuckPosition := PUCKPOS_GRIPPED_AT_TRAY; END_IF;
IF ConvMoveTimer.Q THEN
    DummyDint := MpAlarmXSet(MpLink := gAlarmXCore_Dist, Name := 'Swivel Arm - Motion Blocked');
END_IF;
_p34 := _p33 AND gDistHW.di.SwDrConvPos;
IF _p33 AND gDistHW.di.SwDrConvPos THEN gDistHW.do.SwDrToConv := FALSE; END_IF;
IF _p34 THEN
    MainAutoStep.DIST_SWIVEL_DROP := TRUE;
    MainAutoStep.DIST_SWIVEL_TO_CONV := FALSE;
END_IF;

(* Network 28 *)
_e35(CLK := MainAutoStep.DIST_SWIVEL_DROP);
IF MainMode.Auto AND _e35.Q THEN ModeSwitched := MainCtrl.Input.Par.Mode = DISTCTRL_MANUAL; END_IF;
_p36 := MainMode.Auto AND _e35.Q AND ModeSwitched;
IF MainMode.Auto AND _e35.Q AND ModeSwitched THEN MainMode.Manual := TRUE; END_IF;
IF _p36 THEN MainMode.Auto := FALSE; END_IF;

(* Network 29 *)
IF MainMode.Auto AND MainAutoStep.DIST_SWIVEL_DROP THEN gDistHW.do.EjImpulse := TRUE; END_IF;
DropoffTimer(IN := MainMode.Auto AND MainAutoStep.DIST_SWIVEL_DROP AND gDistHW.do.EjImpulse, PT := DROPOFF_TIMER_DELAY);
IF DropoffTimer.Q THEN
    gDistHW.do.EjImpulse := FALSE;
    DropDone := TRUE;
END_IF;
_p37 := MainMode.Auto AND MainAutoStep.DIST_SWIVEL_DROP AND DropDone;
IF _p37 THEN
    PuckPosition := PUCKPOS_CONV_START;
    MainAutoStep.DIST_SWIVEL_TO_MAG := TRUE;
    MainAutoStep.DIST_SWIVEL_DROP := FALSE;
    DropDone := FALSE;
END_IF;

(* Network 30 *)
_e38(CLK := MainAutoStep.DIST_SWIVEL_TO_MAG);
IF MainMode.Auto AND _e38.Q THEN ModeSwitched := MainCtrl.Input.Par.Mode = DISTCTRL_MANUAL; END_IF;
_p39 := MainMode.Auto AND _e38.Q AND ModeSwitched;
IF MainMode.Auto AND _e38.Q AND ModeSwitched THEN MainMode.Manual := TRUE; END_IF;
IF _p39 THEN MainMode.Auto := FALSE; END_IF;

(* Network 31 *)
_p40 := MainMode.Auto AND MainAutoStep.DIST_SWIVEL_TO_MAG;
IF _p40 THEN gDistHW.do.SwDrToMag := TRUE; END_IF;
_p41 := _p40 AND gDistHW.di.SwDrMagPos;
IF _p40 AND gDistHW.di.SwDrMagPos THEN gDistHW.do.SwDrToMag := FALSE; END_IF;
MagMoveTimer(IN := _p40 AND NOT gDistHW.di.SwDrMagPos, PT := MAG_MOVE_TIMEOUT);
IF _p41 THEN MainAutoStep.DIST_CONV_START := TRUE; END_IF;
IF MagMoveTimer.Q THEN
    DummyDint := MpAlarmXSet(MpLink := gAlarmXCore_Dist, Name := 'Swivel Arm - Motion Blocked');
END_IF;
IF _p41 THEN MainAutoStep.DIST_SWIVEL_TO_MAG := FALSE; END_IF;

(* Network 32 *)
_e42(CLK := MainAutoStep.DIST_CONV_START);
IF MainMode.Auto AND _e42.Q THEN ModeSwitched := MainCtrl.Input.Par.Mode = DISTCTRL_MANUAL; END_IF;
_p43 := MainMode.Auto AND _e42.Q AND ModeSwitched;
IF MainMode.Auto AND _e42.Q AND ModeSwitched THEN MainMode.Manual := TRUE; END_IF;
IF _p43 THEN MainMode.Auto := FALSE; END_IF;

(* Network 33 *)
IF MainMode.Auto AND MainAutoStep.DIST_CONV_START THEN
    OpcUaComm[5] := 1;
    PuckPosition := PUCKPOS_CONV_MID;
    MpAxisBasic_0.MoveVelocity := TRUE;
END_IF;
_p44 := MainMode.Auto AND MainAutoStep.DIST_CONV_START;
IF MainMode.Auto AND MainAutoStep.DIST_CONV_START THEN MainAutoStep.DIST_CONV_MOVING := TRUE; END_IF;
IF _p44 THEN MainAutoStep.DIST_CONV_START := FALSE; END_IF;

(* Network 34 *)
_e45(CLK := MainAutoStep.DIST_CONV_MOVING);
IF MainMode.Auto AND _e45.Q THEN ModeSwitched := MainCtrl.Input.Par.Mode = DISTCTRL_MANUAL; END_IF;
_p46 := MainMode.Auto AND _e45.Q AND ModeSwitched;
IF MainMode.Auto AND _e45.Q AND ModeSwitched THEN MainMode.Manual := TRUE; END_IF;
IF _p46 THEN MainMode.Auto := FALSE; END_IF;

(* Network 35 *)
IF MainMode.Auto AND MainAutoStep.DIST_CONV_MOVING AND gDistHW.di.PuckAtConvEnd THEN
    PuckPosition := PUCKPOS_CONV_END;
END_IF;
_e47(CLK := gDistHW.di.PuckAtConvEnd);
_p48 := MainMode.Auto AND MainAutoStep.DIST_CONV_MOVING AND _e47.Q;
IF _p48 THEN MpAxisBasic_0.MoveVelocity := FALSE; END_IF;
PuckLostTimer(IN := MainMode.Auto AND MainAutoStep.DIST_CONV_MOVING AND NOT gDistHW.di.PuckAtConvEnd, PT := PUCK_LOST_TIMEOUT);
_p49 := MainMode.Auto AND MainAutoStep.DIST_CONV_MOVING;
IF _p48 THEN MainAutoStep.DIST_WAIT := TRUE; END_IF;
IF PuckLostTimer.Q THEN
    DummyDint := MpAlarmXSet(MpLink := gAlarmXCore_Dist, Name := 'Conveyor - Puck Lost');
END_IF;
IF _p48 THEN MainAutoStep.DIST_CONV_MOVING := FALSE; END_IF;
BacklogTimer(IN := _p49 AND NOT gDistHW.di.PuckAtConvEnd, PT := BACKLOG_TIMEOUT);
IF BacklogTimer.Q THEN
    DummyDint := MpAlarmXSet(MpLink := gAlarmXCore_Dist, Name := 'Conveyor - Product Backlog');
END_IF;
IF _p48 THEN
    MainCtrl.Output.Status.DistProductCount := 1 + MainCtrl.Output.Status.DistProductCount;
END_IF;

(* Network 36 *)
_e50(CLK := MainAutoStep.DIST_WAIT);
IF MainMode.Auto AND _e50.Q THEN ModeSwitched := MainCtrl.Input.Par.Mode = DISTCTRL_MANUAL; END_IF;
_p51 := MainMode.Auto AND _e50.Q AND ModeSwitched;
IF MainMode.Auto AND _e50.Q AND ModeSwitched THEN MainMode.Manual := TRUE; END_IF;
IF _p51 THEN MainMode.Auto := FALSE; END_IF;

(* Network 37 *)
IF MainAutoStep.DIST_WAIT THEN
    OpcUaComm[5] := 0;
    SortStateSet := OpcUaComm[6] = 1;
END_IF;
_e52(CLK := SortStateSet);
IF MainAutoStep.DIST_WAIT AND _e52.Q THEN PuckPosition := PUCKPOS_IN_MAG; END_IF;
_p53 := MainAutoStep.DIST_WAIT AND _e52.Q;
IF MainAutoStep.DIST_WAIT AND _e52.Q THEN MainAutoStep.DIST_SWIVEL_TO_HOME := TRUE; END_IF;
IF _p53 THEN MainAutoStep.DIST_WAIT := FALSE; END_IF;

(* Network 38 *)
_e54(CLK := MainAutoStep.DIST_SWIVEL_TO_HOME);
IF MainMode.Auto AND _e54.Q THEN ModeSwitched := MainCtrl.Input.Par.Mode = DISTCTRL_MANUAL; END_IF;
_p55 := MainMode.Auto AND _e54.Q AND ModeSwitched;
IF MainMode.Auto AND _e54.Q AND ModeSwitched THEN MainMode.Manual := TRUE; END_IF;
IF _p55 THEN MainMode.Auto := FALSE; END_IF;

(* Network 39 *)
_p56 := MainMode.Auto AND MainAutoStep.DIST_SWIVEL_TO_HOME;
IF _p56 THEN gDistHW.do.SwDrToConv := TRUE; END_IF;
_p57 := _p56 AND gDistHW.di.SwDrConvPos;
IF _p56 AND gDistHW.di.SwDrConvPos THEN gDistHW.do.SwDrToConv := FALSE; END_IF;
HomeMoveTimer(IN := _p56 AND NOT gDistHW.di.SwDrConvPos, PT := HOME_MOVE_TIMEOUT);
IF _p57 THEN MainAutoStep.DIST_EXTEND_EJECTOR := TRUE; END_IF;
IF HomeMoveTimer.Q THEN
    DummyDint := MpAlarmXSet(MpLink := gAlarmXCore_Dist, Name := 'Swivel Arm - Motion Blocked');
END_IF;
IF _p57 THEN MainAutoStep.DIST_SWIVEL_TO_HOME := FALSE; END_IF;

(* Network 40 *)
IF MpAxisBasic_0.Error THEN Error6057Present := MpAxisBasic_0.Info.Diag.Internal.Code = 6057; END_IF;
MpAxisBasic_0.ErrorReset := MpAxisBasic_0.Error AND Error6057Present;

(* Network 41 *)
MpAxisBasic_0(MpLink := ADR(gAxisBasic), Enable := TRUE, Parameters := ADR(AxisPars), Axis := ADR(gAxisDist), Power := MpAxisBasic_0.Active AND NOT MpAxisBasic_0.Error);

(* Network 42 *)
_p58 := (MainCtrl.Input.Par.Mode = DISTCTRL_MANUAL) AND MainCtrl.Input.Cmd.Ejector.Extend;
IF _p58 THEN
    MainCtrl.Input.Cmd.Ejector.Extend := FALSE;
    MainCtrl.Output.CommandRejected := FALSE;
    CmpPuckInTray := PuckPosition = PUCKPOS_IN_TRAY;
END_IF;
IF _p58 AND CmpPuckInTray THEN
    MainCtrl.Output.CommandRejected := TRUE;
    MainCtrl.Output.RejectionCode := EJECTOR_EXTEND_PUCK_IN_TRAY;
END_IF;
IF _p58 AND gDistHW.di.SwDrMagPos THEN
    MainCtrl.Output.CommandRejected := TRUE;
    MainCtrl.Output.RejectionCode := EJECTOR_EXTEND_SWIVEL_IN_TRAY;
END_IF;
IF _p58 AND gDistHW.di.EjCylExtended THEN
    MainCtrl.Output.CommandRejected := TRUE;
    MainCtrl.Output.RejectionCode := EJECTOR_EXTEND_ALREADY_IN_POS;
END_IF;
IF _p58 AND NOT CmpPuckInTray AND NOT gDistHW.di.EjCylExtended AND NOT gDistHW.di.SwDrMagPos THEN
    gDistHW.do.EjCylPushProduct := TRUE;
END_IF;

(* Network 43 *)
_p59 := (MainCtrl.Input.Par.Mode = DISTCTRL_MANUAL) AND MainCtrl.Input.Cmd.Ejector.Retract;
IF _p59 THEN
    MainCtrl.Input.Cmd.Ejector.Retract := FALSE;
    MainCtrl.Output.CommandRejected := FALSE;
END_IF;
IF _p59 AND gDistHW.di.EjCylRetracted THEN
    MainCtrl.Output.CommandRejected := TRUE;
    MainCtrl.Output.RejectionCode := EJECTOR_RETRACT_ALREADY_IN_POS;
END_IF;
IF _p59 AND NOT gDistHW.di.EjCylRetracted THEN gDistHW.do.EjCylPushProduct := FALSE; END_IF;

(* Network 44 *)
_p60 := (MainCtrl.Input.Par.Mode = DISTCTRL_MANUAL) AND MainCtrl.Input.Cmd.SwivelArm.MoveToMagazine;
IF _p60 THEN
    MainCtrl.Input.Cmd.SwivelArm.MoveToMagazine := FALSE;
    MainCtrl.Output.CommandRejected := FALSE;
    CmpPuckInSwivel := PuckPosition = PUCKPOS_IN_SWIVEL;
    CmpPuckGrippedAtConv := PuckPosition = PUCKPOS_GRIPPED_AT_TRAY;
END_IF;
_t61 := (_p60 AND CmpPuckInSwivel) OR (_p60 AND CmpPuckGrippedAtConv);
IF _t61 THEN
    MainCtrl.Output.CommandRejected := TRUE;
    MainCtrl.Output.RejectionCode := SWIVEL_MOVE_MAG_HOLDING_PUCK;
END_IF;
IF _p60 AND gDistHW.di.SwDrMagPos THEN
    MainCtrl.Output.CommandRejected := TRUE;
    MainCtrl.Output.RejectionCode := SWIVEL_TO_MAG_ALREADY_IN_POS;
END_IF;
_p62 := _p60 AND NOT CmpPuckInSwivel AND NOT CmpPuckGrippedAtConv;
IF _p62 THEN
    gDistHW.do.SwDrToConv := FALSE;
    gDistHW.do.SwDrToMag := TRUE;
END_IF;

(* Network 45 *)
_p63 := (MainCtrl.Input.Par.Mode = DISTCTRL_MANUAL) AND MainCtrl.Input.Cmd.SwivelArm.MoveToConveyor;
IF _p63 THEN
    MainCtrl.Input.Cmd.SwivelArm.MoveToConveyor := FALSE;
    MainCtrl.Output.CommandRejected := FALSE;
END_IF;
IF _p63 AND gDistHW.di.SwDrConvPos THEN
    MainCtrl.Output.CommandRejected := TRUE;
    MainCtrl.Output.RejectionCode := SWIVEL_TO_CONV_ALREADY_IN_POS;
END_IF;
IF _p63 THEN CmpPuckAtConvStart := PuckPosition = PUCKPOS_CONV_START; END_IF;
IF _p63 AND CmpPuckAtConvStart THEN
    MainCtrl.Output.CommandRejected := TRUE;
    MainCtrl.Output.RejectionCode := SWIVEL_MOVE_CONV_PUCK_CONFLICT;
END_IF;
_p64 := _p63 AND NOT gDistHW.di.SwDrConvPos AND NOT CmpPuckAtConvStart;
IF _p64 THEN
    gDistHW.do.SwDrToMag := FALSE;
    gDistHW.do.SwDrToConv := TRUE;
END_IF;

(* Network 46 *)
_p65 := (MainCtrl.Input.Par.Mode = DISTCTRL_MANUAL) AND MainCtrl.Input.Cmd.SwivelArm.VacuumOnImpulse;
IF _p65 THEN MainCtrl.Output.CommandRejected := FALSE; END_IF;
IF _p65 AND gDistHW.di.SwDrMagPos THEN CmpPuckNotInTray := PuckPosition <> PUCKPOS_IN_TRAY; END_IF;
IF _p65 AND gDistHW.di.SwDrConvPos THEN
    CmpPuckNotInConvStart := PuckPosition <> PUCKPOS_CONV_START;
END_IF;
_t66 := ((_p65 AND gDistHW.di.SwDrMagPos AND CmpPuckNotInTray) OR (_p65 AND gDistHW.di.SwDrConvPos AND CmpPuckNotInConvStart)) OR (_p65 AND NOT gDistHW.di.SwDrConvPos AND NOT gDistHW.di.SwDrMagPos);
IF _t66 THEN
    MainCtrl.Input.Cmd.SwivelArm.VacuumOnImpulse := FALSE;
    MainCtrl.Output.CommandRejected := TRUE;
    MainCtrl.Output.RejectionCode := SWIVEL_VAC_ON_NO_PRODUCT;
END_IF;
_p67 := _p65 AND NOT CmpPuckNotInTray AND NOT CmpPuckNotInConvStart;
IF _p67 AND (gDistHW.di.SwDrConvPos OR gDistHW.di.SwDrMagPos) THEN PickupDone := FALSE; END_IF;
_p68 := _p67 AND gDistHW.di.SwDrConvPos;
_p69 := _p67 AND gDistHW.di.SwDrMagPos;
IF _p67 AND (gDistHW.di.SwDrConvPos OR gDistHW.di.SwDrMagPos) THEN gDistHW.do.Vacuum := TRUE; END_IF;
ManualPickupTimer(IN := (_p68 OR _p69) AND gDistHW.do.Vacuum, PT := PICKUP_TIMER_DELAY);
IF ManualPickupTimer.Q THEN
    MainCtrl.Input.Cmd.SwivelArm.VacuumOnImpulse := FALSE;
    gDistHW.do.Vacuum := FALSE;
    PickupDone := TRUE;
END_IF;

(* Network 47 *)
_p70 := (MainCtrl.Input.Par.Mode = DISTCTRL_MANUAL) AND MainCtrl.Input.Cmd.SwivelArm.VacuumOffImpulse;
IF _p70 THEN
    MainCtrl.Output.CommandRejected := FALSE;
    CmpPuckInTransit := PuckPosition = PUCKPOS_IN_SWIVEL;
END_IF;
IF _p70 AND CmpPuckInTransit THEN
    MainCtrl.Output.CommandRejected := TRUE;
    MainCtrl.Output.RejectionCode := SWIVEL_VAC_OFF_PUCK_IN_TRANSIT;
END_IF;
IF _p70 AND NOT CmpPuckInTransit THEN
    DropDone := FALSE;
    gDistHW.do.EjImpulse := TRUE;
END_IF;
ManualDropoffTimer(IN := _p70 AND NOT CmpPuckInTransit AND gDistHW.do.EjImpulse, PT := DROPOFF_TIMER_DELAY);
IF ManualDropoffTimer.Q THEN
    MainCtrl.Input.Cmd.SwivelArm.VacuumOffImpulse := FALSE;
    gDistHW.do.EjImpulse := FALSE;
    DropDone := TRUE;
END_IF;

(* Network 48 *)
_p71 := (MainCtrl.Input.Par.Mode = DISTCTRL_MANUAL) AND MainCtrl.Input.Cmd.Conveyor.JogFwd;
IF _p71 THEN MainCtrl.Output.CommandRejected := FALSE; END_IF;
MpAxisBasic_0.JogPositive := _p71;

(* Network 49 *)
_p72 := (MainCtrl.Input.Par.Mode = DISTCTRL_MANUAL) AND MainCtrl.Input.Cmd.Conveyor.JogBack;
IF _p72 THEN MainCtrl.Output.CommandRejected := FALSE; END_IF;
IF _p72 AND NOT gDistHW.di.ConvStartVacant THEN
    MainCtrl.Output.CommandRejected := TRUE;
    MainCtrl.Output.RejectionCode := CONV_JOG_BACK_PUCK_AT_START;
END_IF;
MpAxisBasic_0.JogNegative := _p72 AND gDistHW.di.ConvStartVacant;

(* Network 50 *)
IF MpAlarmXCheckReaction(MpLink := gAlarmXCore_Dist, Name := 'ErrorReaction') THEN
    SetErrorReaction := TRUE;
END_IF;

(* Network 51 *)
IF SetErrorReaction THEN
    gDistHW.do.EjImpulse := TRUE;
    MainMode.Auto := FALSE;
    gDistHW.do.Vacuum := FALSE;
    gDistHW.do.EjCylPushProduct := FALSE;
    gDistHW.do.SwDrToConv := TRUE;
END_IF;
_p73 := SetErrorReaction;
_p74 := SetErrorReaction AND gDistHW.di.SwDrConvPos;
IF SetErrorReaction AND gDistHW.di.SwDrConvPos THEN SetErrorReaction := FALSE; END_IF;
IF _p74 THEN
    gDistHW.do.EjImpulse := FALSE;
    MainCtrl.Input.Cmd.Home := FALSE;
    gDistHW.do.SwDrToConv := FALSE;
END_IF;
IF _p73 THEN
    gDistHW.do.SwDrToMag := FALSE;
    MpAxisBasic_0.MoveVelocity := FALSE;
    MainAutoStep.DIST_EXTEND_EJECTOR := TRUE;
    MainAutoStep.DIST_CONV_END := FALSE;
    MainAutoStep.DIST_CONV_MOVING := FALSE;
    MainAutoStep.DIST_CONV_START := FALSE;
    MainAutoStep.DIST_INIT := FALSE;
    MainAutoStep.DIST_RETRACT_EJECTOR := FALSE;
    MainAutoStep.DIST_SWIVEL_DROP := FALSE;
    MainAutoStep.DIST_SWIVEL_PICKUP := FALSE;
    MainAutoStep.DIST_SWIVEL_TO_CONV := FALSE;
    MainAutoStep.DIST_SWIVEL_TO_HOME := FALSE;
    MainAutoStep.DIST_SWIVEL_TO_MAG := FALSE;
    MainAutoStep.DIST_SWIVEL_TO_PICKUP := FALSE;
    MainAutoStep.DIST_WAIT := FALSE;
END_IF;
END_PROGRAM
```

#### Exit.ld - Exit code
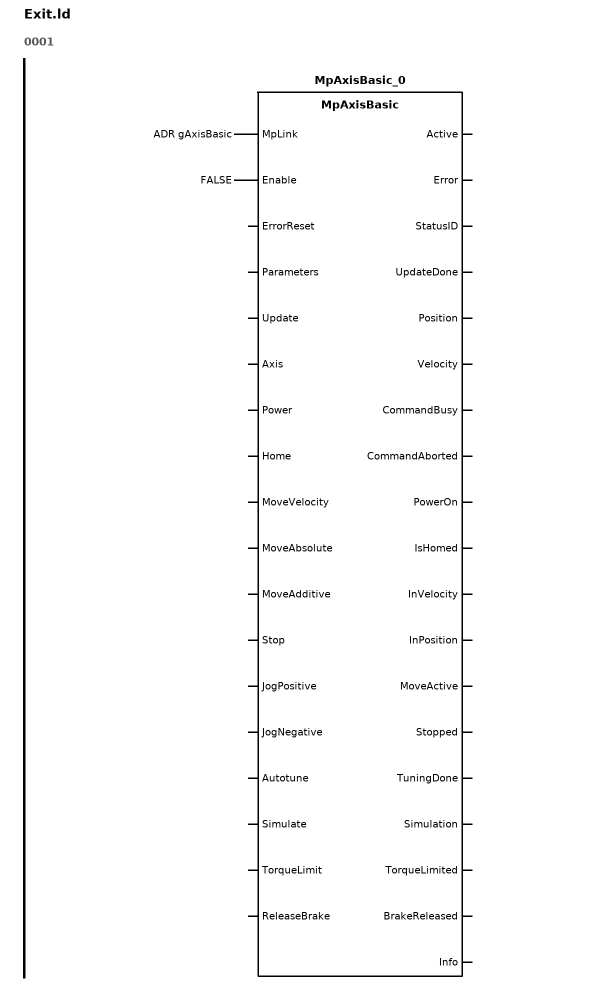
Ladder, written as Structured Text:
```iecst
PROGRAM _EXIT
(* Network 1 *)
MpAxisBasic_0(MpLink := ADR(gAxisBasic), Enable := FALSE);
END_PROGRAM
```

#### Types.typ - Local data types for MainCtrl
```iecst
TYPE
	PuckPosition_Enum :
		(
		PUCKPOS_IN_MAG := 0,
		PUCKPOS_IN_TRANSIT := 1,
		PUCKPOS_IN_TRAY := 2,
		PUCKPOS_GRIPPED_AT_TRAY := 3,
		PUCKPOS_IN_SWIVEL := 4,
		PUCKPOS_GRIPPED_AT_CONV := 5,
		PUCKPOS_CONV_START := 6,
		PUCKPOS_CONV_MID := 7,
		PUCKPOS_CONV_END := 8
		);
	MainAutoStep_typ : 	STRUCT
		DIST_INIT : BOOL;
		DIST_EXTEND_EJECTOR : BOOL;
		DIST_RETRACT_EJECTOR : BOOL;
		DIST_SWIVEL_TO_PICKUP : BOOL;
		DIST_SWIVEL_PICKUP : BOOL;
		DIST_SWIVEL_TO_CONV : BOOL;
		DIST_SWIVEL_DROP : BOOL;
		DIST_SWIVEL_TO_MAG : BOOL;
		DIST_CONV_START : BOOL;
		DIST_CONV_MOVING : BOOL;
		DIST_CONV_END : BOOL;
		DIST_WAIT : BOOL;
		DIST_SWIVEL_TO_HOME : BOOL;
	END_STRUCT;
	MainMode_typ : 	STRUCT
		Auto : BOOL;
		Manual : BOOL;
	END_STRUCT;
END_TYPE
```

#### Variables.var - Local variables for MainCtrl
```iecst
VAR
	MainAutoStep : MainAutoStep_typ := (DIST_INIT:=TRUE,DIST_EXTEND_EJECTOR:=FALSE,DIST_RETRACT_EJECTOR:=FALSE,DIST_SWIVEL_TO_PICKUP:=FALSE,DIST_SWIVEL_PICKUP:=FALSE,DIST_SWIVEL_TO_CONV:=FALSE,DIST_SWIVEL_DROP:=FALSE,DIST_SWIVEL_TO_MAG:=FALSE,DIST_CONV_START:=FALSE,DIST_CONV_MOVING:=FALSE,DIST_CONV_END:=FALSE,DIST_WAIT:=FALSE);
	MainMode : MainMode_typ;
	ModeSwitched : BOOL;
	PickupTimer : TON;
END_VAR
VAR CONSTANT
	PICKUP_TIMER_DELAY : TIME := T#0.5s;
END_VAR
VAR
	PickupDone : BOOL;
	DropDone : BOOL;
	DropoffTimer : TON;
END_VAR
VAR CONSTANT
	DROPOFF_TIMER_DELAY : TIME := T#0.5s;
END_VAR
VAR
	MpAxisBasic_0 : MpAxisBasic; (*Function block for MpAxisBasic*)
	AxisPars : MpAxisBasicParType := (Acceleration:=50.0,Deceleration:=50.0,Velocity:=50.0); (*PArameters for the distributor axis*)
	SortStateSet : BOOL;
	PuckPosition : PuckPosition_Enum := PUCKPOS_IN_MAG; (*tracks the position of the puck through the machine*)
	PuckInTray : BOOL; (*True if a puck is in the magazine tray*)
	CmpPuckInTray : BOOL; (*True if a puck is in the magazine tray*)
	CmpPuckGrippedAtConv : BOOL; (*True if a puck is held by the swivel over the conveyor*)
	CmpPuckInSwivel : BOOL; (*true if puck is held by swivel in transit*)
	CmpPuckAtConvStart : BOOL; (*true if puck is at conveyor start, not held*)
	CmpPuckNotInTray : BOOL; (*true if there is no puck in the magazine tray*)
	CmpPuckNotInConvStart : BOOL; (*true if there is no puck agt conveyor start*)
	ManualPickupTimer : TON; (*Time delay to turn off vacuum pickup*)
	CmpPuckInTransit : BOOL; (*true if puck is moving along the magazine tray*)
	ManualDropoffTimer : TON; (*Time delay to turn off the ejection impulse*)
	SetAlarm : BOOL; (*Intermediate variable for alarm reactions*)
	DummyDint : UDINT; (*Varianle for output of the mpalarmxset function*)
	AutoSelected : BOOL; (*true if automatic mode is selected*)
	SorterInControl : BOOL; (*true if the sorter station is in control of the vis*)
	Error6057Present : BOOL; (*true if error 6057 present*)
	EjectorExtendTimer : TON; (*Timer for ejeectior extend*)
END_VAR
VAR CONSTANT
	EJECTOR_EXTEND_TIMEOUT : TIME := T#5s; (*timeout const for ejector extend*)
END_VAR
VAR
	PickupMoveTimer : TON; (*Timeout timer for swivel arm movement*)
END_VAR
VAR CONSTANT
	PICKUP_MOVE_TIMEOUT : TIME := T#5s; (*Timeout timer for swivel arm movement - constant*)
END_VAR
VAR
	ConvMoveTimer : TON; (*Timeout timer for swivel arm movement*)
END_VAR
VAR CONSTANT
	CONV_MOVE_TIMEOUT : TIME := T#5s; (*Timeout timer for swivel arm movement - constant*)
END_VAR
VAR
	MagMoveTimer : TON; (*Timeout timer for swivel arm movement*)
END_VAR
VAR CONSTANT
	MAG_MOVE_TIMEOUT : TIME := T#5s; (*Timeout timer for swivel arm movement - constant*)
END_VAR
VAR
	HomeMoveTimer : TON; (*Timeout timer for swivel arm movement*)
END_VAR
VAR CONSTANT
	HOME_MOVE_TIMEOUT : TIME := T#5s; (*Timeout timer for swivel arm movement - constant*)
END_VAR
VAR
	PuckLostTimer : TON; (*Timeout timer for conveyor*)
END_VAR
VAR CONSTANT
	PUCK_LOST_TIMEOUT : TIME := T#15s; (*timeout timer constant for conveyor*)
END_VAR
VAR
	BacklogTimer : TON; (*timeout timer for part passing end sensor*)
END_VAR
VAR CONSTANT
	BACKLOG_TIMEOUT : TIME := T#10s; (*constant for timeout timer for part passing end sensor*)
END_VAR
VAR
	SetErrorReaction : BOOL; (*Intermediate variable used for error reactions*)
	StartAutoRequested : BOOL; (*Start auto is requested*)
	ControlHeld : BOOL; (*True if distributor has control of the vis*)
END_VAR
```

#### ActivateVacuum.ld - not listed in the package file held
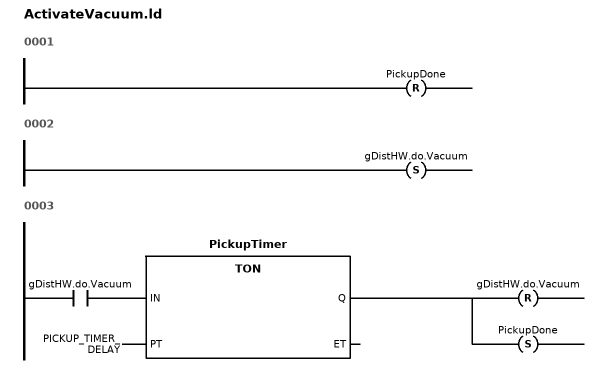
Ladder, written as Structured Text:
```iecst
ACTION ActivateVacuum:
(* Network 1 *)
PickupDone := FALSE;

(* Network 2 *)
gDistHW.do.Vacuum := TRUE;

(* Network 3 *)
PickupTimer(IN := gDistHW.do.Vacuum, PT := PICKUP_TIMER_DELAY);
IF PickupTimer.Q THEN
    gDistHW.do.Vacuum := FALSE;
    PickupDone := TRUE;
END_IF;
END_ACTION
```

#### DeactivateVacuum.ld - not listed in the package file held
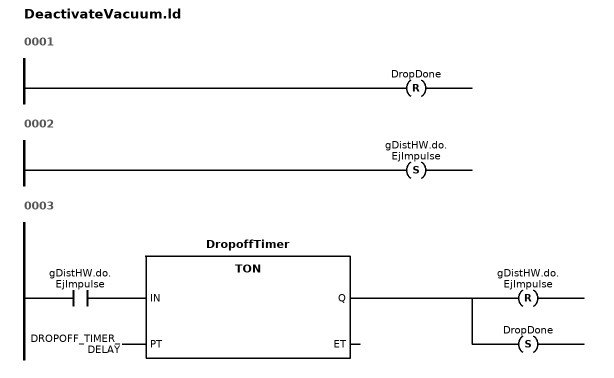
Ladder, written as Structured Text:
```iecst
ACTION DeactivateVacuum:
(* Network 1 *)
DropDone := FALSE;

(* Network 2 *)
gDistHW.do.EjImpulse := TRUE;

(* Network 3 *)
DropoffTimer(IN := gDistHW.do.EjImpulse, PT := DROPOFF_TIMER_DELAY);
IF DropoffTimer.Q THEN
    gDistHW.do.EjImpulse := FALSE;
    DropDone := TRUE;
END_IF;
END_ACTION
```

### Stations.typ - not listed in the package file held
```iecst
(*Ejector Station Interface Structures*)

TYPE
	Ejector_typ : {REDUND_UNREPLICABLE} 	STRUCT  (*Interface for Ejector station. Accessed by the Distributor MainCtrl Program.*)
		Input : {REDUND_UNREPLICABLE} EjectorInput_typ; (*Input for Ejector Station, contains Commands and Parameters.*)
		Output : {REDUND_UNREPLICABLE} EjectorOutput_typ; (*Output for Ejector Station, contains Statuses(e.g. cylinder position) and information regarding which commands are allowed at any given time*)
	END_STRUCT;
	EjectorInput_typ : {REDUND_UNREPLICABLE} 	STRUCT  (*Ejector Input*)
		Cmd : {REDUND_UNREPLICABLE} EjectorCmd_typ; (*Commands for the Ejector Station. Includes a command to run a full ejector cycle, as well as commands for finer control of the station, to be used during manual mode.*)
		Par : {REDUND_UNREPLICABLE} EjectorPar_typ; (*Parameters for the Ejector Station.*)
	END_STRUCT;
	EjectorPar_typ : 	STRUCT  (*Ejector Parameters*)
		Placeholder : USINT; (*Placeholder for parameters*)
	END_STRUCT;
	EjectorCmd_typ : 	STRUCT  (*Ejector Commands*)
		ExtendEjector : BOOL := FALSE; (*Command to extend the ejector cylinder*)
		RetractEjector : BOOL := FALSE; (*Command to retract the ejector cylinder*)
		RunCycle : BOOL := FALSE; (*Command to run one full cycle of the ejector station*)
		ErrorReset : BOOL := FALSE; (*Command to reset station errors*)
		Home : BOOL := FALSE; (*Command to home the station*)
	END_STRUCT;
	EjectorOutput_typ : 	STRUCT  (*Ejector Output*)
		Status : EjectorStatus_typ; (*Status of the ejector station. Contains information about the ejector cylinder position, state of the magazine (empty,not empty), and whether there is an error on the station*)
		CommandRejected : BOOL := FALSE; (*True if the issued command is not allowed. The RejectionCode is set accordingly to provide feedback on why a command may not be allowed.*)
		RejectionCode : EjectorRejectionCode_Enum; (*Provides feedback on why a command may not be allowed at a given time.*)
	END_STRUCT;
	EjectorRejectionCode_Enum :
		( (*Information about which command was rejected, and why*)
		EJECTOR_CYL_ALREADY_EXTENDED := 0,
		EJECTOR_CYL_ALREADY_RETRACTED,
		EJECTOR_STN_ALREADY_HOMED
		);
	EjectorStatus_typ : 	STRUCT  (*Ejector Status*)
		EjectorExtended : BOOL; (*True if the ejector cylinder is fully extended*)
		EjectorRetracted : BOOL; (*True if the ejector cylinder is fully retracted*)
		Error : BOOL; (*True if the station is in an error state*)
		ErrorID : EjectorErrorID_Enum; (*Container for error information*)
		IsHomed : BOOL; (*True if the station is in the home position*)
		CycleDone : BOOL;
	END_STRUCT;
	EjectorErrorID_Enum :
		( (*Information about Error status of the Ejector Task*)
		EJECTOR_ERROR_EXTEND_BLOCKED
		);
END_TYPE

(*Ejector Station Interface Structures*)

TYPE
	SwivelArm_typ : {REDUND_UNREPLICABLE} 	STRUCT  (*Interface for Ejector station. Accessed by the Distributor MainCtrl Program.*)
		Input : {REDUND_UNREPLICABLE} SwivelArmInput_typ; (*Input for Ejector Station, contains Commands and Parameters.*)
		Output : {REDUND_UNREPLICABLE} SwivelArmOutput_typ; (*Output for Ejector Station, contains Statuses(e.g. cylinder position) and information regarding which commands are allowed at any given time*)
	END_STRUCT;
	SwivelArmInput_typ : {REDUND_UNREPLICABLE} 	STRUCT  (*Ejector Input*)
		Cmd : {REDUND_UNREPLICABLE} SwivelArmCmd_typ; (*Commands for the Ejector Station. Includes a command to run a full ejector cycle, as well as commands for finer control of the station, to be used during manual mode.*)
		Par : {REDUND_UNREPLICABLE} SwivelArmPar_typ; (*Parameters for the Ejector Station.*)
	END_STRUCT;
	SwivelArmPar_typ : 	STRUCT  (*Ejector Parameters*)
		Placeholder : USINT; (*Placeholder for parameters*)
	END_STRUCT;
	SwivelArmCmd_typ : 	STRUCT  (*Ejector Commands*)
		MoveToMagazine : BOOL := FALSE; (*Command to extend the ejector cylinder*)
		MoveToConveyor : BOOL := FALSE; (*Command to retract the ejector cylinder*)
		ActivateVacuum : BOOL := FALSE; (*Command to run one full cycle of the ejector station*)
		DeactivateVacuum : BOOL := FALSE; (*Command to reset station errors*)
		Home : BOOL;
		RunCycle : BOOL;
		ErrorReset : BOOL := FALSE; (*Command to home the station*)
	END_STRUCT;
	SwivelArmOutput_typ : 	STRUCT  (*Ejector Output*)
		Status : SwivelArmStatus_typ; (*Status of the ejector station. Contains information about the ejector cylinder position, state of the magazine (empty,not empty), and whether there is an error on the station*)
		CommandRejected : BOOL := FALSE; (*True if the issued command is not allowed. The RejectionCode is set accordingly to provide feedback on why a command may not be allowed.*)
		RejectionCode : SwivelArmRejectionCode_Enum; (*Provides feedback on why a command may not be allowed at a given time.*)
	END_STRUCT;
	SwivelArmRejectionCode_Enum :
		( (*Information about which command was rejected, and why*)
		SWIVEL_ALREADY_AT_CONV := 0,
		SWIVEL_ALREADY_AT_MAG,
		SWIVEL_VAC_ALREADY_INACTIVE,
		SWIVEL_VAC_ALREADY_ACTIVE,
		SWIVEL_ALREADY_HOMED
		);
	SwivelArmStatus_typ : 	STRUCT  (*Ejector Status*)
		AtMagazine : BOOL; (*True if the ejector cylinder is fully extended*)
		AtConveyor : BOOL; (*True if the ejector cylinder is fully retracted*)
		VacuumOn : BOOL; (*True if the station is in an error state*)
		ErrorID : SwivelArmErrorID_Enum; (*Container for error information*)
		IsHomed : BOOL; (*True if the station is in the home position*)
		CycleDone : BOOL;
	END_STRUCT;
	SwivelArmErrorID_Enum :
		( (*Information about Error status of the Ejector Task*)
		SWIVEL_ERROR
		);
END_TYPE

(*SwivelArm Station Interface Structures*)

TYPE
	Conveyor_typ : {REDUND_UNREPLICABLE} 	STRUCT  (*Interface for Ejector station. Accessed by the Distributor MainCtrl Program.*)
		Input : {REDUND_UNREPLICABLE} ConveyorInput_typ; (*Input for Ejector Station, contains Commands and Parameters.*)
		Output : {REDUND_UNREPLICABLE} ConveyorOutput_typ; (*Output for Ejector Station, contains Statuses(e.g. cylinder position) and information regarding which commands are allowed at any given time*)
	END_STRUCT;
	ConveyorInput_typ : {REDUND_UNREPLICABLE} 	STRUCT  (*Ejector Input*)
		Cmd : {REDUND_UNREPLICABLE} ConveyorCmd_typ; (*Commands for the Ejector Station. Includes a command to run a full ejector cycle, as well as commands for finer control of the station, to be used during manual mode.*)
		Par : {REDUND_UNREPLICABLE} ConveyorPar_typ; (*Parameters for the Ejector Station.*)
	END_STRUCT;
	ConveyorPar_typ : 	STRUCT  (*Ejector Parameters*)
		Accel : REAL := 5000;
		Speed : REAL := 2000; (*Placeholder for parameters*)
		Decel : REAL := 5000;
	END_STRUCT;
	ConveyorCmd_typ : 	STRUCT  (*Ejector Commands*)
		JogForward : BOOL := FALSE; (*Command to run one full cycle of the ejector station*)
		JogBackward : BOOL := FALSE; (*Command to reset station errors*)
		RunCycle : BOOL;
		ErrorReset : BOOL := FALSE; (*Command to home the station*)
	END_STRUCT;
	ConveyorOutput_typ : 	STRUCT  (*Ejector Output*)
		Status : ConveyorStatus_typ; (*Status of the ejector station. Contains information about the ejector cylinder position, state of the magazine (empty,not empty), and whether there is an error on the station*)
		CommandRejected : BOOL := FALSE; (*True if the issued command is not allowed. The RejectionCode is set accordingly to provide feedback on why a command may not be allowed.*)
		RejectionCode : ConveyorRejectionCode_Enum; (*Provides feedback on why a command may not be allowed at a given time.*)
	END_STRUCT;
	ConveyorRejectionCode_Enum :
		( (*Information about which command was rejected, and why*)
		CONV_PART_AT_START
		);
	ConveyorStatus_typ : 	STRUCT  (*Ejector Status*)
		AtMagazine : BOOL; (*True if the ejector cylinder is fully extended*)
		AtConveyor : BOOL; (*True if the ejector cylinder is fully retracted*)
		VacuumOn : BOOL; (*True if the station is in an error state*)
		ErrorID : ConveyorErrorID_typ; (*Container for error information*)
		IsHomed : BOOL; (*True if the station is in the home position*)
		CycleDone : BOOL;
	END_STRUCT;
	ConveyorErrorID_typ :
		( (*Information about Error status of the Ejector Task*)
		CONV_ERROR
		);
END_TYPE
```
